# B&R Automation Studio project Soiled_PLC (part 5)

#### 12_sp2Cyclic.ab
```automation-basic
PROGRAM _CYCLIC
	(* cyclic program *)

;---------------------------------------
;Sequence 8 - SP8 Single point 2 D[912]
;---------------------------------------

;Inputs

O_SelectLine[11]          = FALSE
O_SelectLine[12]          = FALSE ;YB10
O_SelectLine[13]          = FALSE ;YB10
EnableRel.PC[2]           = FALSE
MySeq                     = 40
MyBag                     = 156
MyTransBag                = 158

I_BagatBuffer	          = RequestRel.PC[1]

O_Reset                   = FALSE

Alarm[MySeq].Name 			= 0
Alarm[MySeq].Bag			= MyTransBag
Alarm[MySeq].Beacon		    = TRUE
Alarm[MySeq].Extra			= 0
Alarm[MySeq].Time			= 5000

;Setup Sequence
STEP = D[900 + MySeq]
;Setup Pulse contact
PLS = (STEP <> LASTSTEP)
LASTSTEP = STEP

;Sequence
;Step 0 - Disabled
IF (STEP = 0) THEN
	;Disabled
ENDIF

;clear data
TON_10ms((STEP = 1),100,Reset,ResetET)
IF (STEP = 1) THEN
	O_Reset = TRUE
	IF (Reset = TRUE)AND (Bag[MyTransBag].Cat = 0) THEN
		D[900 + MySeq] = 2
	ENDIF
	IF Reset THEN
		Alarm[MySeq].Time			= 5
		Alarm[MySeq].Name 	= almBagDataError
	ENDIF
ENDIF

;Wait SLU1 request and destination clear
TON_10ms(I_BagatBuffer,300,BagAtBuffer,BagAtBufferET)
IF (STEP = 2) THEN
	IF (Bag[MyBag].Cat >0) AND (Bag[MyBag].Dst >0) AND RequestRel.PC[1] THEN
		IF (Line[Bag[MyBag].Dst].Space > 0) AND (Bag[MyBag].Dst > 10) AND (Bag[MyBag].Dst < 14) AND (Line[Bag[MyBag].Dst].Clear) AND (Bag[Line[Bag[MyBag].Dst].LastBag].Cat = 0) THEN
			Dest = Bag[MyBag].Dst
			C[Dest]        = 0
			D[900 + MySeq] = 3
		ENDIF

	ENDIF
ENDIF

		;Open buffer to release a bag to svc 1
IF (STEP = 3) THEN
	EnableRel.PC[2] = TRUE
	O_SelectLine[Dest] = TRUE
	IF PLS THEN
		IF (Bag[MyBag].Cat>0) AND (Bag[MyTransBag].Cat = 0)	THEN

			Bag[MyTransBag]     = Bag[MyBag]
			Bag[MyBag]          = Bag[0]
		ENDIF
	ENDIF
	IF (Dest = 13) THEN
		IF (Bag[MyTransBag].Cat>0) AND (Bag[159].Cat=0) AND X[4].X16 THEN
			Bag[159] = Bag[MyTransBag]
			Bag[MyTransBag] = Bag[0]
		ENDIF
		IF Line[Dest].Trip THEN
			IF ((Bag[73].Cat = 0) AND (Bag[159].Cat>0)) THEN
				Bag[159].Dst = 0
				Bag[73]      = Bag[159]
				Bag[159]     = Bag[0]
			ENDIF
			D[900 + MySeq] = 1
		ENDIF
    ELSE IF (Dest > 10) AND (Dest < 13) THEN
			IF Line[Dest].Trip THEN
				Bag[MyTransBag].Dst     = 0
				Bag[Line[Dest].LastBag] = Bag[MyTransBag]
				Bag[MyTransBag]         = Bag[0]
				D[900 + MySeq] = 1
		ENDIF

	ENDIF

	Alarm[MySeq].Name 	= almBagNotArrived
ENDIF

;select svc 2 point
IF (STEP = 4) THEN
O_SelectSVC2 = TRUE

	IF Line[18].Trip THEN
		IF (Bag[221].Cat > 0) AND (Bag[222].Cat= 0) THEN
			Bag[222] = Bag[221]
			Bag[221] = Bag[0]
		ENDIF
		D[900 + MySeq] = 1
	ENDIF
	Alarm[MySeq].Name 	= almBagNotArrived
ENDIF

;Outputs

Y[5].Y08 = O_SelectLine[11]
Y[5].Y09 = O_SelectLine[12]
Y[5].Y10 = O_Reset OR O_SelectLine[13]

;Alarms
TimerAlarm.IN 	= NOT PLS AND (Alarm[MySeq].Name > 0)
TimerAlarm.PT 	= Alarm[MySeq].Time
TimerAlarm FUB TON_10ms()
Alarm[MySeq].On 	= TimerAlarm.Q
Alarm[MySeq].ET 	= TimerAlarm.ET

;Outputs
;Y[6].Y07 = O_SelectPointSVC1
;Y[6].Y08 = O_SelectPointSVC2
END_PROGRAM
```

#### 12_sp2.var
```iecst
VAR RETAIN
	STEP : UINT;
	PLS : BOOL;
	LASTSTEP : UINT;
END_VAR
VAR
	TimerAlarm : TON_10ms;
	I_BagAtBuffer : BOOL;
	O_OpenBuffer : BOOL;
	SDC2BufferFullET : TIME;
	SDC2BufferFull : BOOL;
	SettledBufferET : TIME;
	SettledBuffer : BOOL;
	O_OpenSP2BufferStop : BOOL;
	O_SelectPoint : BOOL;
	SP2BufferFull : BOOL;
	SP2BufferFullET : UDINT;
	ParingLoopEnabled : BOOL;
	BagInLoopHasDest : BOOL;
	BagAtBuffer : BOOL;
	SettledBufferSVC1 : BOOL;
	SettledBufferSVC1ET : UDINT;
	SettledBufferSVC2 : BOOL;
	SettledBufferSVC2ET : UDINT;
	O_SelectPointSVC1 : BOOL;
	O_SelectPointSVC2 : BOOL;
	Reset : BOOL;
	ResetET : UDINT;
	I_BagatBuffer : BOOL;
	BagAtBufferET : UDINT;
	Alernate : USINT;
	I_BagAtSVC1BufferStop : BOOL;
	O_SVC1BufferStop : BOOL;
	I_BagAtSVC2BufferStop : BOOL;
	O_SVC2BufferStop : BOOL;
	O_SelectSVC1 : BOOL;
	O_SelectSVC2 : BOOL;
	MySeq : USINT;
	MyBag : USINT;
	MyTransBag : INT;
	Dest : INT;
	O_SelectLine : ARRAY[0..13] OF BOOL;
	O_Reset : BOOL;
END_VAR
```

### Program Logical/Sequences/10ms/41_cp8 (IEC) - * SP2 Empty bags from SDC1/2

#### 12_sp2.var
```iecst
VAR RETAIN
	STEP : UINT;
	PLS : BOOL;
	LASTSTEP : UINT;
END_VAR
VAR
	TimerAlarm : TON_10ms;
	I_BagAtBuffer : ARRAY[0..3] OF BOOL;
	O_OpenBuffer : BOOL;
	SDC2BufferFullET : TIME;
	SDC2BufferFull : BOOL;
	SettledBufferET : TIME;
	SettledBuffer : ARRAY[0..3] OF BOOL;
	O_OpenSP2BufferStop : BOOL;
	O_SelectPoint : BOOL;
	SP2BufferFull : BOOL;
	SP2BufferFullET : UDINT;
	ParingLoopEnabled : BOOL;
	BagInLoopHasDest : BOOL;
	O_OpenSDC1BufferStop : BOOL;
	BagSettledAtBuffer : BOOL;
	BagSettledAtBufferET : UDINT;
	Alternator : USINT;
	I_OnLineA : BOOL;
	I_TiltA : BOOL;
	I_TiltB : BOOL;
	I_Bagout : BOOL;
	O_OpenBufferStop : BOOL;
	O_SelectLineA : BOOL;
	O_SelectLineB : BOOL;
	O_OpenStops : BOOL;
	O_TiltCylinder : BOOL;
	O_OperatePusher : BOOL;
	PointReset : BOOL;
	PointResetET : UDINT;
	BagAtTilt : BOOL;
	BagAtTiltET : UDINT;
	TiltDown : BOOL;
	TiltDownET : UDINT;
	TiltUp : BOOL;
	TiltUpET : UDINT;
	NotFull : BOOL;
	NotFullET : UDINT;
	Pushed : BOOL;
	SBSN1 : BOOL;
	SBSN1ET : UDINT;
	RequirePusherET : UDINT;
	PushedET : UDINT;
	I_BagAtBufferStop : BOOL;
	O_SP7ToSVC1 : BOOL;
	O_SP7ToSIC3 : BOOL;
	SDC1EmptyBufferFull : BOOL;
	SDC1EmptyBufferFullET : UDINT;
	Reset : BOOL;
	ResetET : UDINT;
	ResetPoint : BOOL;
	I_SDC1EmptyBagAtBuffer : BOOL;
	O_ResetPoints : BOOL;
	BagSettledSDC1Buffer : BOOL;
	BagSettledSDC1BufferET : UDINT;
	BagSettledSDC2Buffer : BOOL;
	BagSettledSDC2BufferET : UDINT;
	MySeq : USINT;
	BagSettledBufferET : ARRAY[0..3] OF UDINT;
	Alt : USINT;
	O_SelectCDC4 : BOOL;
	O_SelectStraight : BOOL;
	O_SelectCDC3 : BOOL;
	O_SelectCPI4 : BOOL;
	O_SelectCP6 : BOOL;
	O_Reset : BOOL;
END_VAR
```

#### 12_sp2Cyclic.ab
```automation-basic
PROGRAM _CYCLIC
	(* cyclic program *)

;---------------------------------------
;Sequence 12 - SP2 Single point 2 D[912]
;---------------------------------------

;Inputs

I_BagAtBuffer[1]		= Request.DCEmptyRelease[3]
I_BagAtBuffer[2]		= X[10].X04
I_BagAtBuffer[3]		= X[10].X05

MySeq                   = 41

Alarm[MySeq].Name 			= 0
Alarm[MySeq].Bag			= 10013
Alarm[MySeq].Beacon		= TRUE
Alarm[MySeq].Extra			= 0
Alarm[MySeq].Time			= 3000

Enable.DCEmptyRelease[3]    = FALSE

O_SelectCDC3                = FALSE
O_SelectCPI4                = FALSE
O_SelectCP6                 = FALSE
O_Reset                     = FALSE

;Setup Sequence
STEP = D[900 + MySeq]
;Setup Pulse contact
PLS = (STEP <> LASTSTEP)
LASTSTEP = STEP

;Sequence
;Step 0 - Disabled
IF (STEP = 0) THEN
	;Disabled
ENDIF

;reset points
TON_10ms((STEP = 1),200,Reset,ResetET)
IF (STEP = 1) THEN
	O_Reset = NOT Reset
	IF (Line[42].Clear) AND Reset  THEN
		D[900 + MySeq] = 2
	ENDIF
	ELSE

ENDIF

;check which bag is ready
TON_10ms(I_BagAtBuffer[1],200,SettledBuffer[1],BagSettledBufferET[1])
TON_10ms(I_BagAtBuffer[2],200,SettledBuffer[2],BagSettledBufferET[2])
TON_10ms(I_BagAtBuffer[3],200,SettledBuffer[3],BagSettledBufferET[3])
IF (STEP = 2) THEN
	IF (Line[42].Clear) AND NOT Y[4].Y15 AND NOT X[8].X08 THEN
		;Alt = Alt + 1
		;IF (Alt > 2) THEN
		;	Alt = 0
		;ENDIF
		IF SettledBuffer[1]  THEN
			C[42]          = 0
		    D[900 + MySeq] = 3
		ELSE IF SettledBuffer[2]  THEN
			C[42]          = 0
			D[900 + MySeq] = 4
		ELSE IF SettledBuffer[3] AND (D[8]>0)  THEN
			C[42]          = 0
			D[900 + MySeq] = 5
		ENDIF
	ENDIF
ENDIF

;Bag at line
IF (STEP = 3) THEN
	O_SelectCDC3 = TRUE
	Enable.DCEmptyRelease[3] = TRUE
	IF (Line[42].Trip = TRUE) THEN
		D[900 + MySeq] = 1
	ENDIF
	Alarm[MySeq].Name 	  = almBagNotArrived
ENDIF

;Bag at line
IF (STEP = 4) THEN
	O_SelectCP6 = TRUE
	IF (Line[42].Trip = TRUE) THEN
		D[900 + MySeq] = 1
	ENDIF
	Alarm[MySeq].Name 	  = almBagNotArrived
ENDIF

;Bag at line
IF (STEP = 5) THEN
	O_SelectCPI4 = TRUE
	IF (Line[42].Trip = TRUE) THEN
		D[900 + MySeq] = 1
	ENDIF
	Alarm[MySeq].Name 	  = almBagNotArrived
ENDIF
;Alarms
TimerAlarm.IN 	= NOT PLS AND (Alarm[MySeq].Name > 0)
TimerAlarm.PT 	= Alarm[MySeq].Time
TimerAlarm FUB TON_10ms()
Alarm[MySeq].On 	= TimerAlarm.Q
Alarm[MySeq].ET 	= TimerAlarm.ET

;Outputs
Y[9].Y09 = O_SelectCDC3
Y[8].Y03 = O_SelectCP6
Y[8].Y04 = O_SelectCPI4
Y[8].Y08 = O_Reset

END_PROGRAM
```

### Program Logical/Sequences/10ms/42_cp9 (IEC) - * SP2 Empty bags from SDC1/2

#### 12_sp2.var
```iecst
VAR RETAIN
	STEP : UINT;
	PLS : BOOL;
	LASTSTEP : UINT;
END_VAR
VAR
	TimerAlarm : TON_10ms;
	I_BagAtBuffer : ARRAY[0..3] OF BOOL;
	O_OpenBuffer : BOOL;
	SDC2BufferFullET : TIME;
	SDC2BufferFull : BOOL;
	SettledBufferET : TIME;
	SettledBuffer : ARRAY[0..3] OF BOOL;
	O_OpenSP2BufferStop : BOOL;
	O_SelectPoint : BOOL;
	SP2BufferFull : BOOL;
	SP2BufferFullET : UDINT;
	ParingLoopEnabled : BOOL;
	BagInLoopHasDest : BOOL;
	O_OpenSDC1BufferStop : BOOL;
	BagSettledAtBuffer : BOOL;
	BagSettledAtBufferET : UDINT;
	Alternator : USINT;
	I_OnLineA : BOOL;
	I_TiltA : BOOL;
	I_TiltB : BOOL;
	I_Bagout : BOOL;
	O_OpenBufferStop : BOOL;
	O_SelectLineA : BOOL;
	O_SelectLineB : BOOL;
	O_OpenStops : BOOL;
	O_TiltCylinder : BOOL;
	O_OperatePusher : BOOL;
	PointReset : BOOL;
	PointResetET : UDINT;
	BagAtTilt : BOOL;
	BagAtTiltET : UDINT;
	TiltDown : BOOL;
	TiltDownET : UDINT;
	TiltUp : BOOL;
	TiltUpET : UDINT;
	NotFull : BOOL;
	NotFullET : UDINT;
	Pushed : BOOL;
	SBSN1 : BOOL;
	SBSN1ET : UDINT;
	RequirePusherET : UDINT;
	PushedET : UDINT;
	I_BagAtBufferStop : BOOL;
	O_SP7ToSVC1 : BOOL;
	O_SP7ToSIC3 : BOOL;
	SDC1EmptyBufferFull : BOOL;
	SDC1EmptyBufferFullET : UDINT;
	Reset : BOOL;
	ResetET : UDINT;
	ResetPoint : BOOL;
	I_SDC1EmptyBagAtBuffer : BOOL;
	O_ResetPoints : BOOL;
	BagSettledSDC1Buffer : BOOL;
	BagSettledSDC1BufferET : UDINT;
	BagSettledSDC2Buffer : BOOL;
	BagSettledSDC2BufferET : UDINT;
	MySeq : USINT;
	BagSettledBufferET : ARRAY[0..3] OF UDINT;
	Alt : USINT;
	O_SelectCDC4 : BOOL;
	O_SelectStraight : BOOL;
	O_Reset : BOOL;
	O_SelectCLU1 : BOOL;
	O_SelectCLU2 : BOOL;
END_VAR
```

#### 12_sp2Cyclic.ab
```automation-basic
PROGRAM _CYCLIC
	(* cyclic program *)

;---------------------------------------
;Sequence 12 - SP2 Single point 2 D[912]
;---------------------------------------

;Inputs

I_BagAtBuffer[1]		= X[8].X16
;I_BagAtBuffer[2]		= X[9].X14

MySeq                   = 42

Alarm[MySeq].Name 			= 0
Alarm[MySeq].Bag			= 10005
Alarm[MySeq].Beacon		= TRUE
Alarm[MySeq].Extra			= 0
Alarm[MySeq].Time			= 3000

O_SelectCLU1                = FALSE
O_SelectCLU2                = FALSE

;Setup Sequence
STEP = D[900 + MySeq]
;Setup Pulse contact
PLS = (STEP <> LASTSTEP)
LASTSTEP = STEP

;Sequence
;Step 0 - Disabled
IF (STEP = 0) THEN
	;Disabled
ENDIF

;reset points
TON_10ms((STEP = 1),200,Reset,ResetET)
IF (STEP = 1) THEN
	O_Reset = NOT Reset
	IF (Reset)  THEN
		D[900 + MySeq] = 2
	ENDIF
	ELSE

ENDIF

;check which bag is ready
TON_10ms(I_BagAtBuffer[1],200,SettledBuffer[1],BagSettledBufferET[1])

IF (STEP = 2) THEN
	IF SettledBuffer[1] THEN
		Alt = Alt + 1
		IF (Alt > 2) THEN
			Alt = 0
		ENDIF
		IF SettledBuffer[1] AND (Alt = 1) AND Line[35].Clear THEN
			C[35]          = 0
		    D[900 + MySeq] = 3
		ELSE IF SettledBuffer[1] AND (Alt = 2) AND Line[36].Clear THEN
			C[36]          = 0
			D[900 + MySeq] = 4
		ENDIF
	ENDIF
ENDIF

;Bag at line
IF (STEP = 3) THEN
	O_SelectCLU1 = TRUE
	IF (Line[35].Trip = TRUE) THEN
		D[900 + MySeq] = 1
	ENDIF
	Alarm[MySeq].Name 	  = almBagNotArrived
ENDIF

;Bag at line
IF (STEP = 4) THEN
	O_SelectCLU2 = TRUE
	IF (Line[36].Trip = TRUE) THEN
		D[900 + MySeq] = 1
	ENDIF
	Alarm[MySeq].Name 	  = almBagNotArrived
ENDIF

;Alarms
TimerAlarm.IN 	= NOT PLS AND (Alarm[MySeq].Name > 0)
TimerAlarm.PT 	= Alarm[MySeq].Time
TimerAlarm FUB TON_10ms()
Alarm[MySeq].On 	= TimerAlarm.Q
Alarm[MySeq].ET 	= TimerAlarm.ET

;Outputs
Y[8].Y05 = O_SelectCLU1
Y[8].Y06 = O_SelectCLU2
Y[8].Y07 = O_SelectCLU1 OR O_SelectCLU2
END_PROGRAM
```

### Program Logical/Sequences/10ms/43_cp12 (IEC) - * SP2 Empty bags from SDC1/2

#### 12_sp2.var
```iecst
VAR RETAIN
	STEP : UINT;
	PLS : BOOL;
	LASTSTEP : UINT;
END_VAR
VAR
	TimerAlarm : TON_10ms;
	I_BagAtBuffer : ARRAY[0..3] OF BOOL;
	O_OpenBuffer : BOOL;
	SDC2BufferFullET : TIME;
	SDC2BufferFull : BOOL;
	SettledBufferET : TIME;
	SettledBuffer : ARRAY[0..3] OF BOOL;
	O_OpenSP2BufferStop : BOOL;
	O_SelectPoint : BOOL;
	SP2BufferFull : BOOL;
	SP2BufferFullET : UDINT;
	ParingLoopEnabled : BOOL;
	BagInLoopHasDest : BOOL;
	O_OpenSDC1BufferStop : BOOL;
	BagSettledAtBuffer : BOOL;
	BagSettledAtBufferET : UDINT;
	Alternator : USINT;
	I_OnLineA : BOOL;
	I_TiltA : BOOL;
	I_TiltB : BOOL;
	I_Bagout : BOOL;
	O_OpenBufferStop : BOOL;
	O_SelectLineA : BOOL;
	O_SelectLineB : BOOL;
	O_OpenStops : BOOL;
	O_TiltCylinder : BOOL;
	O_OperatePusher : BOOL;
	PointReset : BOOL;
	PointResetET : UDINT;
	BagAtTilt : BOOL;
	BagAtTiltET : UDINT;
	TiltDown : BOOL;
	TiltDownET : UDINT;
	TiltUp : BOOL;
	TiltUpET : UDINT;
	NotFull : BOOL;
	NotFullET : UDINT;
	Pushed : BOOL;
	SBSN1 : BOOL;
	SBSN1ET : UDINT;
	RequirePusherET : UDINT;
	PushedET : UDINT;
	I_BagAtBufferStop : BOOL;
	O_SP7ToSVC1 : BOOL;
	O_SP7ToSIC3 : BOOL;
	SDC1EmptyBufferFull : BOOL;
	SDC1EmptyBufferFullET : UDINT;
	Reset : BOOL;
	ResetET : UDINT;
	ResetPoint : BOOL;
	I_SDC1EmptyBagAtBuffer : BOOL;
	O_ResetPoints : BOOL;
	BagSettledSDC1Buffer : BOOL;
	BagSettledSDC1BufferET : UDINT;
	BagSettledSDC2Buffer : BOOL;
	BagSettledSDC2BufferET : UDINT;
	MySeq : USINT;
	BagSettledBufferET : ARRAY[0..3] OF UDINT;
	Alt : USINT;
	O_SelectCDC4 : BOOL;
	O_SelectStraight : BOOL;
	O_SelectCIC5 : BOOL;
	O_SelectCDC6 : BOOL;
	O_Reset : BOOL;
	O_SelectCDC5 : BOOL;
	O_SelectCDC7 : BOOL;
	O_SelectCDC8 : BOOL;
	O_SelectCDC9 : BOOL;
	Dest : USINT;
END_VAR
```

#### 12_sp2Cyclic.ab
```automation-basic
PROGRAM _CYCLIC
	(* cyclic program *)

;---------------------------------------
;Sequence 12 - SP2 Single point 2 D[912]
;---------------------------------------

;Inputs

I_BagAtBuffer[1]		= RequestRel.IC[5]
;I_BagAtBuffer[2]		= X[9].X14

MySeq                   = 43

Alarm[MySeq].Name 			= 0
Alarm[MySeq].Bag			= 166
Alarm[MySeq].Beacon		= TRUE
Alarm[MySeq].Extra			= 0
Alarm[MySeq].Time			= 3000

O_SelectCDC7                = FALSE
O_SelectCDC8               = FALSE
O_SelectCDC9                = FALSE
EnableRel.IC[5]             = FALSE
O_Reset                     = FALSE

;Setup Sequence
STEP = D[900 + MySeq]
;Setup Pulse contact
PLS = (STEP <> LASTSTEP)
LASTSTEP = STEP

;Sequence
;Step 0 - Disabled
IF (STEP = 0) THEN
	;Disabled
ENDIF

;reset points
TON_10ms((STEP = 1),200,Reset,ResetET)
IF (STEP = 1) THEN
	O_Reset = TRUE
	IF Reset  THEN
		D[900 + MySeq] = 2
	ENDIF
	ELSE

ENDIF

;check which bag is ready
TON_10ms(I_BagAtBuffer[1],200,SettledBuffer[1],BagSettledBufferET[1])

IF (STEP = 2) THEN
	IF SettledBuffer[1] AND (D[43] >0)  THEN
		Dest = Bag[152].Dst
		IF (Dest = 17) AND Line[17].Clear AND (Bag[92].Cat = 0) THEN
			C[17]                  = 0
			D[900 + MySeq] = 3
        ELSE IF (Dest = 18) AND Line[18].Clear AND (Bag[97].Cat = 0) THEN
			C[18]                  = 0
			D[900 + MySeq] = 4
		 ELSE IF (Dest = 19) AND Line[26].Clear AND (Bag[151].Cat = 0) THEN
			C[26]                  = 0
			D[900 + MySeq] = 5
		ENDIF
	ENDIF
ENDIF

;Bag at line
IF (STEP = 3) THEN
	O_SelectCDC7 = TRUE
	EnableRel.IC[5] = TRUE
;	IF (Bag[152].Cat>0) AND (Bag[166].Cat = 0) THEN
;		Bag[166] = Bag[152]
;		Bag[152] = Bag[0]
;	ENDIF
	IF Line[17].Trip THEN
		IF (Bag[166].Cat > 0) AND (Bag[92].Cat = 0) THEN
			Bag[92] = Bag[166]
			Bag[166]= Bag[0]

		ENDIF
			D[900 + MySeq] = 1
	ENDIF
	Alarm[MySeq].Name 	  = almBagNotArrived
ENDIF

;Bag at line
IF (STEP = 4) THEN
	O_SelectCDC8 = TRUE
	EnableRel.IC[5] = TRUE
;	IF (Bag[152].Cat>0) AND (Bag[166].Cat = 0) THEN
;		Bag[166] = Bag[152]
;		Bag[152] = Bag[0]
;	ENDIF
	IF (Line[18].Trip = TRUE) THEN
		IF (Bag[166].Cat > 0) AND (Bag[97].Cat = 0) THEN
			Bag[97] = Bag[166]
			Bag[166]= Bag[0]

		ENDIF
		D[900 + MySeq] = 1
	ENDIF
	Alarm[MySeq].Name 	  = almBagNotArrived
ENDIF

IF (STEP = 5) THEN
	O_SelectCDC9 = TRUE
	EnableRel.IC[5] = TRUE
;	IF (Bag[152].Cat>0) AND (Bag[166].Cat = 0) THEN
;		Bag[166] = Bag[152]
;		Bag[152] = Bag[0]
;	ENDIF
	IF (Line[26].Trip = TRUE) THEN
		IF (Bag[166].Cat > 0) AND (Bag[151].Cat = 0) THEN
			Bag[166].Dst = 0
			Bag[151]       = Bag[166]
			Bag[166]       = Bag[0]

		ENDIF
		D[900 + MySeq] = 1
	ENDIF
	Alarm[MySeq].Name 	  = almBagNotArrived
ENDIF

;Alarms
TimerAlarm.IN 	= NOT PLS AND (Alarm[MySeq].Name > 0)
TimerAlarm.PT 	= Alarm[MySeq].Time
TimerAlarm FUB TON_10ms()
Alarm[MySeq].On 	= TimerAlarm.Q
Alarm[MySeq].ET 	= TimerAlarm.ET

;Outputs
Y[1].Y13 = O_SelectCDC7
Y[2].Y03 = O_SelectCDC8
Y[10].Y03 = O_Reset OR O_SelectCDC9
Y[10].Y04 = O_Reset OR O_SelectCDC9
END_PROGRAM
```

### Program Logical/Sequences/10ms/44_cpr2 (IEC, version 1.00.2) - *Pressure Relief

#### pr.st - Implementation code
```iecst
(********************************************************************
 * COPYRIGHT --
 ********************************************************************
 * Program: pr
 * File: pr.st
 * Author: treamsbottom
 * Created: July 16, 2015
 ********************************************************************
 * Implementation of program pr
 ********************************************************************)

PROGRAM _INIT
//Configuration
mySeq						:= 44;	//Sequence number
myIO						:= 9;
myZone						:= 0;
myRelLine					:= 28;
myBag						:= 0; //Buffer Bag
bufferSettleTime			:= 300;

myOutBag 					:= Line[myRelLine].LastBag;
END_PROGRAM

PROGRAM _CYCLIC
//Inputs
i_bagAtBuffer				:= X[myIO].X08;

i_bagAtBufferOut 		:= FALSE; // Any Single bag buffer out IO.
i_bufferOutOpen			:= FALSE;

o_openBuffer	:= FALSE;

IF (myBag = 0) THEN
	Alarm[mySeq].Bag	:= mySeq + 10000;
ELSE
	Alarm[mySeq].Bag	:= myBag;
END_IF;

Alarm[mySeq].Name 		:= 0;
Alarm[mySeq].Beacon		:= TRUE;
Alarm[mySeq].Extra		:= 0;
Alarm[mySeq].Time		:= 3000;

//Setup Sequence
step := D[900 + mySeq];
//Setup Pulse contact
pls := (step <> lastStep);
lastStep := step;

//Sequence
IF (step = 0) THEN
	//Disabled
END_IF;

//Bag Settled at buffer
ton_10ms_SettledBuffer(IN:= i_bagAtBuffer, PT:= bufferSettleTime);
IF (step = 1) THEN
	IF ton_10ms_SettledBuffer.Q AND NOT Std.HaltSysZone[myZone]THEN
		IF Line[myRelLine].Clear AND NOT i_bagAtBufferOut AND NOT i_bufferOutOpen AND NOT Line[myRelLine].Trip THEN
			IF (myBag = 0) THEN
				C[myRelLine] := 0;
				D[900 + mySeq] := 2;
			ELSIF (Bag[myBag].Cat > 0) AND (Bag[myOutBag].Cat = 0) THEN
				C[myRelLine] := 0;
				D[900 + mySeq] := 2;
			ELSIF (Bag[myBag].Cat = 0) THEN
				Alarm[mySeq].Name := ALM_BAG_DATA_ERROR;
				Alarm[mySeq].Time := 0;
			ELSIF (Bag[myOutBag].Cat > 0) THEN
				Alarm[mySeq].Name := ALM_BAG_DATA_ERROR;
				Alarm[mySeq].Bag := myOutBag;
				Alarm[mySeq].Time := 0;
			END_IF;
		ELSIF Line[myRelLine].Trip THEN
			Alarm[mySeq].Name := ALM_SWITCH_FAULT; //Trip is stuck on
			Alarm[mySeq].Time := 500;
		END_IF;
	ELSIF (myBag > 0) AND (Bag[myBag].Cat > 0) THEN
		Alarm[mySeq].Name := ALM_BAG_NOT_SETTLED;
	END_IF;
END_IF;

IF (step = 2) THEN
	dataValid := ((myBag = 0) OR ((Bag[myBag].Cat > 0) AND (Bag[myOutBag].Cat = 0)));
	o_openBuffer :=  dataValid;
	IF dataValid THEN
		IF Line[myRelLine].Trip THEN
			IF (myBag > 0) THEN
				Bag[myOutBag] := Bag[myBag];
				Bag[myBag]  := Bag[0];
			END_IF;
			D[900 + mySeq] := 1;
		END_IF;
		Alarm[mySeq].Name := ALM_BAG_NOT_RELEASED;
	ELSIF (myBag > 0) THEN
		IF (Bag[myBag].Cat = 0) THEN
			Alarm[mySeq].Name := ALM_BAG_DATA_ERROR;
			Alarm[mySeq].Time := 0;
		ELSIF (Bag[myOutBag].Cat > 0) THEN
			Alarm[mySeq].Name := ALM_BAG_DATA_ERROR;
			Alarm[mySeq].Bag := myOutBag;
			Alarm[mySeq].Time := 0;
		END_IF;
	END_IF;
END_IF;

//-----------------------------------
//PLC Outputs - adjust TO suit system
//-----------------------------------

Y[myIO].Y08 := o_openBuffer;

//Alarms
timerAlarm(IN := NOT pls AND (Alarm[mySeq].Name > 0),PT:= Alarm[mySeq].Time);

Alarm[mySeq].On 	:= timerAlarm.Q;
Alarm[mySeq].ET 	:= timerAlarm.ET;

END_PROGRAM
```

### Program Logical/Sequences/10ms/45_cpr3 (IEC) - *Pressure Relief

#### pr.st
```iecst
(********************************************************************
 * COPYRIGHT --
 ********************************************************************
 * Program: pr
 * File: pr.st
 * Author: treamsbottom
 * Created: July 16, 2015
 ********************************************************************
 * Implementation of program pr
 ********************************************************************)

PROGRAM _INIT
//Configuration
mySeq						:= 45;	//Sequence number
myIO						:= 9;
myZone						:= 0;
myRelLine					:= 39;
myBag						:= 0; //Buffer Bag
bufferSettleTime			:= 300;

myOutBag 					:= Line[myRelLine].LastBag;
END_PROGRAM

PROGRAM _CYCLIC
//Inputs
i_bagAtBuffer				:= X[myIO].X12;

i_bagAtBufferOut 		:= FALSE; // Any Single bag buffer out IO.
i_bufferOutOpen			:= FALSE;

o_openBuffer	:= FALSE;

IF (myBag = 0) THEN
	Alarm[mySeq].Bag	:= mySeq + 10000;
ELSE
	Alarm[mySeq].Bag	:= myBag;
END_IF;

Alarm[mySeq].Name 		:= 0;
Alarm[mySeq].Beacon		:= TRUE;
Alarm[mySeq].Extra		:= 0;
Alarm[mySeq].Time		:= 3000;

//Setup Sequence
step := D[900 + mySeq];
//Setup Pulse contact
pls := (step <> lastStep);
lastStep := step;

//Sequence
IF (step = 0) THEN
	//Disabled
END_IF;

//Bag Settled at buffer
ton_10ms_SettledBuffer(IN:= i_bagAtBuffer, PT:= bufferSettleTime);
IF (step = 1) THEN
	IF ton_10ms_SettledBuffer.Q AND NOT Std.HaltSysZone[myZone]THEN
		IF Line[myRelLine].Clear AND NOT i_bagAtBufferOut AND NOT i_bufferOutOpen AND NOT Line[myRelLine].Trip THEN
			IF (myBag = 0) THEN
				C[myRelLine] := 0;
				D[900 + mySeq] := 2;
			ELSIF (Bag[myBag].Cat > 0) AND (Bag[myOutBag].Cat = 0) THEN
				C[myRelLine] := 0;
				D[900 + mySeq] := 2;
			ELSIF (Bag[myBag].Cat = 0) THEN
				Alarm[mySeq].Name := ALM_BAG_DATA_ERROR;
				Alarm[mySeq].Time := 0;
			ELSIF (Bag[myOutBag].Cat > 0) THEN
				Alarm[mySeq].Name := ALM_BAG_DATA_ERROR;
				Alarm[mySeq].Bag := myOutBag;
				Alarm[mySeq].Time := 0;
			END_IF;
		ELSIF Line[myRelLine].Trip THEN
			Alarm[mySeq].Name := ALM_SWITCH_FAULT; //Trip is stuck on
			Alarm[mySeq].Time := 500;
		END_IF;
	ELSIF (myBag > 0) AND (Bag[myBag].Cat > 0) THEN
		Alarm[mySeq].Name := ALM_BAG_NOT_SETTLED;
	END_IF;
END_IF;

IF (step = 2) THEN
	dataValid := ((myBag = 0) OR ((Bag[myBag].Cat > 0) AND (Bag[myOutBag].Cat = 0)));
	o_openBuffer :=  dataValid;
	IF dataValid THEN
		IF Line[myRelLine].Trip THEN
			IF (myBag > 0) THEN
				Bag[myOutBag] := Bag[myBag];
				Bag[myBag]  := Bag[0];
			END_IF;
			D[900 + mySeq] := 1;
		END_IF;
		Alarm[mySeq].Name := ALM_BAG_NOT_RELEASED;
	ELSIF (myBag > 0) THEN
		IF (Bag[myBag].Cat = 0) THEN
			Alarm[mySeq].Name := ALM_BAG_DATA_ERROR;
			Alarm[mySeq].Time := 0;
		ELSIF (Bag[myOutBag].Cat > 0) THEN
			Alarm[mySeq].Name := ALM_BAG_DATA_ERROR;
			Alarm[mySeq].Bag := myOutBag;
			Alarm[mySeq].Time := 0;
		END_IF;
	END_IF;
END_IF;

//-----------------------------------
//PLC Outputs - adjust TO suit system
//-----------------------------------

Y[9].Y12 := o_openBuffer;

//Alarms
timerAlarm(IN := NOT pls AND (Alarm[mySeq].Name > 0),PT:= Alarm[mySeq].Time);

Alarm[mySeq].On 	:= timerAlarm.Q;
Alarm[mySeq].ET 	:= timerAlarm.ET;

END_PROGRAM
```

### Program Logical/Sequences/10ms/46_cpr4 (IEC) - *Pressure Relief

#### pr.st
```iecst
(********************************************************************
 * COPYRIGHT --
 ********************************************************************
 * Program: pr
 * File: pr.st
 * Author: treamsbottom
 * Created: July 16, 2015
 ********************************************************************
 * Implementation of program pr
 ********************************************************************)

PROGRAM _INIT
//Configuration
mySeq						:= 46;	//Sequence number
myIO						:= 220;
myZone						:= 0;
myRelLine					:= 40;
myBag						:= 0; //Buffer Bag
bufferSettleTime			:= 300;

myOutBag 					:= Line[myRelLine].LastBag;
END_PROGRAM

PROGRAM _CYCLIC
//Inputs
i_bagAtBuffer				:= X[11].X10;

i_bagAtBufferOut 		:= FALSE; // Any Single bag buffer out IO.
i_bufferOutOpen			:= FALSE;

o_openBuffer	:= FALSE;

IF (myBag = 0) THEN
	Alarm[mySeq].Bag	:= mySeq + 10000;
ELSE
	Alarm[mySeq].Bag	:= myBag;
END_IF;

Alarm[mySeq].Name 		:= 0;
Alarm[mySeq].Beacon		:= TRUE;
Alarm[mySeq].Extra		:= 0;
Alarm[mySeq].Time		:= 3000;

//Setup Sequence
step := D[900 + mySeq];
//Setup Pulse contact
pls := (step <> lastStep);
lastStep := step;

//Sequence
IF (step = 0) THEN
	//Disabled
END_IF;

//Bag Settled at buffer
ton_10ms_SettledBuffer(IN:= i_bagAtBuffer, PT:= bufferSettleTime);
IF (step = 1) THEN
	IF ton_10ms_SettledBuffer.Q AND NOT Std.HaltSysZone[myZone]THEN
		IF Line[myRelLine].Clear AND NOT i_bagAtBufferOut AND NOT i_bufferOutOpen AND NOT Line[myRelLine].Trip THEN
			IF (myBag = 0) THEN
				C[myRelLine] := 0;
				D[900 + mySeq] := 2;
			ELSIF (Bag[myBag].Cat > 0) AND (Bag[myOutBag].Cat = 0) THEN
				C[myRelLine] := 0;
				D[900 + mySeq] := 2;
			ELSIF (Bag[myBag].Cat = 0) THEN
				Alarm[mySeq].Name := ALM_BAG_DATA_ERROR;
				Alarm[mySeq].Time := 0;
			ELSIF (Bag[myOutBag].Cat > 0) THEN
				Alarm[mySeq].Name := ALM_BAG_DATA_ERROR;
				Alarm[mySeq].Bag := myOutBag;
				Alarm[mySeq].Time := 0;
			END_IF;
		ELSIF Line[myRelLine].Trip THEN
			Alarm[mySeq].Name := ALM_SWITCH_FAULT; //Trip is stuck on
			Alarm[mySeq].Time := 500;
		END_IF;
	ELSIF (myBag > 0) AND (Bag[myBag].Cat > 0) THEN
		Alarm[mySeq].Name := ALM_BAG_NOT_SETTLED;
	END_IF;
END_IF;

IF (step = 2) THEN
	dataValid := ((myBag = 0) OR ((Bag[myBag].Cat > 0) AND (Bag[myOutBag].Cat = 0)));
	o_openBuffer :=  dataValid;
	IF dataValid THEN
		IF Line[myRelLine].Trip THEN
			IF (myBag > 0) THEN
				Bag[myOutBag] := Bag[myBag];
				Bag[myBag]  := Bag[0];
			END_IF;
			D[900 + mySeq] := 1;
		END_IF;
		Alarm[mySeq].Name := ALM_BAG_NOT_RELEASED;
	ELSIF (myBag > 0) THEN
		IF (Bag[myBag].Cat = 0) THEN
			Alarm[mySeq].Name := ALM_BAG_DATA_ERROR;
			Alarm[mySeq].Time := 0;
		ELSIF (Bag[myOutBag].Cat > 0) THEN
			Alarm[mySeq].Name := ALM_BAG_DATA_ERROR;
			Alarm[mySeq].Bag := myOutBag;
			Alarm[mySeq].Time := 0;
		END_IF;
	END_IF;
END_IF;

//-----------------------------------
//PLC Outputs - adjust TO suit system
//-----------------------------------

Y[10].Y10 := o_openBuffer;

//Alarms
timerAlarm(IN := NOT pls AND (Alarm[mySeq].Name > 0),PT:= Alarm[mySeq].Time);

Alarm[mySeq].On 	:= timerAlarm.Q;
Alarm[mySeq].ET 	:= timerAlarm.ET;

END_PROGRAM
```

- Standard_Sequence_Pressure_Relief_ENG.docx (binary file, 203948 bytes)
### Program Logical/Sequences/10ms/47_cpr1 (IEC) - *Pressure Relief

#### pr.var
```iecst
(********************************************************************
 * COPYRIGHT --
 ********************************************************************
 * Program: pr
 * File: pr.var
 * Author: treamsbottom
 * Created: July 16, 2015
 ********************************************************************
 * Local variables of program pr
 ********************************************************************)
VAR
	mySeq : UINT;
	myIO : UINT;
	myZone : UINT;
	myRelLine : UINT;
	myBag : UINT;
	i_bagAtBuffer : BOOL;
	i_bagAtBufferOut : BOOL;
	i_bufferOutOpen : BOOL;
	o_openBuffer : BOOL;
	step : UINT;
	pls : BOOL;
	timerAlarm : TON_10ms;
END_VAR
VAR RETAIN
	lastStep : UINT;
END_VAR
VAR
	bufferSettleTime : UDINT;
	ton_10ms_SettledBuffer : TON_10ms;
	myOutBag : UINT;
	dataValid : BOOL;
END_VAR
```

#### pr.st
```iecst
(********************************************************************
 * COPYRIGHT --
 ********************************************************************
 * Program: pr
 * File: pr.st
 * Author: treamsbottom
 * Created: July 16, 2015
 ********************************************************************
 * Implementation of program pr
 ********************************************************************)

PROGRAM _INIT
//Configuration
mySeq						:= 47;	//Sequence number
myIO						:= 9;
myZone						:= 0;
myRelLine					:= 43;
myBag						:= 0; //Buffer Bag
bufferSettleTime			:= 300;

myOutBag 					:= Line[myRelLine].LastBag;
END_PROGRAM

PROGRAM _CYCLIC
//Inputs
i_bagAtBuffer				:= X[myIO].X03;

i_bagAtBufferOut 		:= FALSE; // Any Single bag buffer out IO.
i_bufferOutOpen			:= FALSE;

o_openBuffer	:= FALSE;

IF (myBag = 0) THEN
	Alarm[mySeq].Bag	:= mySeq + 10000;
ELSE
	Alarm[mySeq].Bag	:= myBag;
END_IF;

Alarm[mySeq].Name 		:= 0;
Alarm[mySeq].Beacon		:= TRUE;
Alarm[mySeq].Extra		:= 0;
Alarm[mySeq].Time		:= 3000;

//Setup Sequence
step := D[900 + mySeq];
//Setup Pulse contact
pls := (step <> lastStep);
lastStep := step;

//Sequence
IF (step = 0) THEN
	//Disabled
END_IF;

//Bag Settled at buffer
ton_10ms_SettledBuffer(IN:= i_bagAtBuffer, PT:= bufferSettleTime);
IF (step = 1) THEN
	IF ton_10ms_SettledBuffer.Q AND NOT Std.HaltSysZone[myZone]THEN
		IF Line[myRelLine].Clear AND NOT i_bagAtBufferOut AND NOT i_bufferOutOpen AND NOT Line[myRelLine].Trip THEN
			IF (myBag = 0) THEN
				C[myRelLine] := 0;
				D[900 + mySeq] := 2;
			ELSIF (Bag[myBag].Cat > 0) AND (Bag[myOutBag].Cat = 0) THEN
				C[myRelLine] := 0;
				D[900 + mySeq] := 2;
			ELSIF (Bag[myBag].Cat = 0) THEN
				Alarm[mySeq].Name := ALM_BAG_DATA_ERROR;
				Alarm[mySeq].Time := 0;
			ELSIF (Bag[myOutBag].Cat > 0) THEN
				Alarm[mySeq].Name := ALM_BAG_DATA_ERROR;
				Alarm[mySeq].Bag := myOutBag;
				Alarm[mySeq].Time := 0;
			END_IF;
		ELSIF Line[myRelLine].Trip THEN
			Alarm[mySeq].Name := ALM_SWITCH_FAULT; //Trip is stuck on
			Alarm[mySeq].Time := 500;
		END_IF;
	ELSIF (myBag > 0) AND (Bag[myBag].Cat > 0) THEN
		Alarm[mySeq].Name := ALM_BAG_NOT_SETTLED;
	END_IF;
END_IF;

IF (step = 2) THEN
	dataValid := ((myBag = 0) OR ((Bag[myBag].Cat > 0) AND (Bag[myOutBag].Cat = 0)));
	o_openBuffer :=  dataValid;
	IF dataValid THEN
		IF Line[myRelLine].Trip THEN
			IF (myBag > 0) THEN
				Bag[myOutBag] := Bag[myBag];
				Bag[myBag]  := Bag[0];
			END_IF;
			D[900 + mySeq] := 1;
		END_IF;
		Alarm[mySeq].Name := ALM_BAG_NOT_RELEASED;
	ELSIF (myBag > 0) THEN
		IF (Bag[myBag].Cat = 0) THEN
			Alarm[mySeq].Name := ALM_BAG_DATA_ERROR;
			Alarm[mySeq].Time := 0;
		ELSIF (Bag[myOutBag].Cat > 0) THEN
			Alarm[mySeq].Name := ALM_BAG_DATA_ERROR;
			Alarm[mySeq].Bag := myOutBag;
			Alarm[mySeq].Time := 0;
		END_IF;
	END_IF;
END_IF;

//-----------------------------------
//PLC Outputs - adjust TO suit system
//-----------------------------------

Y[5].Y16 := o_openBuffer;

//Alarms
timerAlarm(IN := NOT pls AND (Alarm[mySeq].Name > 0),PT:= Alarm[mySeq].Time);

Alarm[mySeq].On 	:= timerAlarm.Q;
Alarm[mySeq].ET 	:= timerAlarm.ET;

END_PROGRAM
```

### Program Logical/Sequences/10ms/48_cp6 (IEC) - * SP2 Empty bags from SDC1/2

#### 12_sp2.var
```iecst
VAR RETAIN
	STEP : UINT;
	PLS : BOOL;
	LASTSTEP : UINT;
END_VAR
VAR
	TimerAlarm : TON_10ms;
	I_BagAtBuffer : ARRAY[0..3] OF BOOL;
	O_OpenBuffer : BOOL;
	SDC2BufferFullET : TIME;
	SDC2BufferFull : BOOL;
	SettledBufferET : TIME;
	SettledBuffer : ARRAY[0..3] OF BOOL;
	O_OpenSP2BufferStop : BOOL;
	O_SelectPoint : BOOL;
	SP2BufferFull : BOOL;
	SP2BufferFullET : UDINT;
	ParingLoopEnabled : BOOL;
	BagInLoopHasDest : BOOL;
	O_OpenSDC1BufferStop : BOOL;
	BagSettledAtBuffer : BOOL;
	BagSettledAtBufferET : UDINT;
	Alternator : USINT;
	I_OnLineA : BOOL;
	I_TiltA : BOOL;
	I_TiltB : BOOL;
	I_Bagout : BOOL;
	O_OpenBufferStop : BOOL;
	O_SelectLineA : BOOL;
	O_SelectLineB : BOOL;
	O_OpenStops : BOOL;
	O_TiltCylinder : BOOL;
	O_OperatePusher : BOOL;
	PointReset : BOOL;
	PointResetET : UDINT;
	BagAtTilt : BOOL;
	BagAtTiltET : UDINT;
	TiltDown : BOOL;
	TiltDownET : UDINT;
	TiltUp : BOOL;
	TiltUpET : UDINT;
	NotFull : BOOL;
	NotFullET : UDINT;
	Pushed : BOOL;
	SBSN1 : BOOL;
	SBSN1ET : UDINT;
	RequirePusherET : UDINT;
	PushedET : UDINT;
	I_BagAtBufferStop : BOOL;
	O_SP7ToSVC1 : BOOL;
	O_SP7ToSIC3 : BOOL;
	SDC1EmptyBufferFull : BOOL;
	SDC1EmptyBufferFullET : UDINT;
	Reset : BOOL;
	ResetET : UDINT;
	ResetPoint : BOOL;
	I_SDC1EmptyBagAtBuffer : BOOL;
	O_ResetPoints : BOOL;
	BagSettledSDC1Buffer : BOOL;
	BagSettledSDC1BufferET : UDINT;
	BagSettledSDC2Buffer : BOOL;
	BagSettledSDC2BufferET : UDINT;
	MySeq : USINT;
	BagSettledBufferET : ARRAY[0..3] OF UDINT;
	Alt : USINT;
	O_SelectCDC4 : BOOL;
	O_SelectStraight : BOOL;
	O_SelectCDC1 : BOOL;
	O_SelectCDC2 : BOOL;
END_VAR
```

#### 12_sp2Cyclic.ab
```automation-basic
PROGRAM _CYCLIC
	(* cyclic program *)

;---------------------------------------
;Sequence 12 - SP2 Single point 2 D[912]
;---------------------------------------

;Inputs

I_BagAtBuffer[1]		= X[5].X14
I_BagAtBuffer[2]		= X[5].X15

MySeq                   = 48

Alarm[MySeq].Name 			= 0
Alarm[MySeq].Bag			= 10001
Alarm[MySeq].Beacon		= TRUE
Alarm[MySeq].Extra			= 0
Alarm[MySeq].Time			= 3000

O_SelectCDC1                = FALSE
O_SelectCDC2             = FALSE

;Setup Sequence
STEP = D[900 + MySeq]
;Setup Pulse contact
PLS = (STEP <> LASTSTEP)
LASTSTEP = STEP

;Sequence
;Step 0 - Disabled
IF (STEP = 0) THEN
	;Disabled
ENDIF

;reset points
TON_10ms((STEP = 1),200,Reset,ResetET)
IF (STEP = 1) THEN

	IF (Line[47].Clear)  THEN
		D[900 + MySeq] = 2
	ENDIF
	ELSE

ENDIF

;check which bag is ready
TON_10ms(I_BagAtBuffer[1],200,SettledBuffer[1],BagSettledBufferET[1])
TON_10ms(I_BagAtBuffer[2],200,SettledBuffer[2],BagSettledBufferET[2])
IF (STEP = 2) THEN
	IF (Line[47].Clear) THEN
		Alt = Alt + 1
		IF (Alt > 2) THEN
			Alt = 0
		ENDIF
		IF SettledBuffer[1] AND (Alt = 1) THEN
			C[47]          = 0
		    D[900 + MySeq] = 3
		ELSE IF SettledBuffer[2] AND (Alt = 2) THEN
			C[47]          = 0
			D[900 + MySeq] = 4
		ENDIF
	ENDIF
ENDIF

;Bag at line
IF (STEP = 3) THEN
	O_SelectCDC1 = TRUE
	IF (Line[47].Trip = TRUE) THEN
		D[900 + MySeq] = 1
	ENDIF
	Alarm[MySeq].Name 	  = almBagNotArrived
ENDIF

;Bag at line
IF (STEP = 4) THEN
	O_SelectCDC2 = TRUE
	IF (Line[47].Trip = TRUE) THEN
		D[900 + MySeq] = 1
	ENDIF
	Alarm[MySeq].Name 	  = almBagNotArrived
ENDIF

;Alarms
TimerAlarm.IN 	= NOT PLS AND (Alarm[MySeq].Name > 0)
TimerAlarm.PT 	= Alarm[MySeq].Time
TimerAlarm FUB TON_10ms()
Alarm[MySeq].On 	= TimerAlarm.Q
Alarm[MySeq].ET 	= TimerAlarm.ET

;Outputs
Y[5].Y12 = O_SelectCDC1
Y[5].Y13 = O_SelectCDC2
END_PROGRAM
```

### Program Logical/Sequences/10ms/9_sic1_ref (IEC) - * SIC1 Incline Conveyor 1

#### 9_sic1Cyclic.ab
```automation-basic
PROGRAM _CYCLIC
	(* cyclic program *)

;---------------------------------------------------
;Sequence 12 - SIC1 Soiled Incline Conveyor 1 D[909]
;---------------------------------------------------

;Inputs

I_BagAtBuffer			= X[8].X06
I_PaddleInPosition		= X[6].X15
I_BagInIncline			= X[6].X14

O_OpenBufferStop		= FALSE
O_RunMotor 				= FALSE

I_BagAtOutgoingBuffer	= FALSE
O_OutgoingBufferOpen	= FALSE

Enable.IC[1]			= FALSE
O_SelectSDC1            = FALSE
O_SelectSDC2            = FALSE

Alarm[9].Name 			= 0
Alarm[9].Bag			= 287
Alarm[9].Beacon			= TRUE
Alarm[9].Extra			= 0
Alarm[9].Time			= 3000

;Setup Sequence
STEP = D[909]
;Setup Pulse contact
PLS = (STEP <> LASTSTEP)
LASTSTEP = STEP

;Sequence
;Step 0 - Disabled
IF (STEP = 0) THEN
	;Disabled
ENDIF

;Run Incline until paddle in position
IF (STEP = 1) THEN
	O_RunMotor = NOT I_PaddleInPosition
	IF I_PaddleInPosition THEN
		D[909] = 2
	ENDIF
	IF NOT Std.EStop THEN
		Alarm[9].Name = almSwitchFault
	ENDIF
ENDIF

;Wait for at buffer
TON_10ms(I_BagAtBuffer,300,BagAtBuffer,BagAtBufferET)
IF (STEP = 2) THEN
	IF (BagAtBuffer AND (Bag[240].Cat > 0) AND NOT Std.HaltSys) THEN
		D[909] = 3
	ENDIF
	IF (Bag[240].Cat > 0) AND NOT I_BagAtBuffer THEN
		Alarm[9].Name 	= almBagNotAtProx
		Alarm[9].Bag	= 240
	ELSE IF (Bag[240].Cat = 0) AND I_BagAtBuffer THEN
		Alarm[9].Name 	= almBagNotShownOnScreen
		Alarm[9].Bag	= 240
	ENDIF
ENDIF

;Open Buffer stop
IF (STEP = 3) THEN
	O_OpenBufferStop 	= TRUE
	Enable.IC[1]		= (NOT I_BagInIncline AND (Bag[240].Cat = 0))
	IF I_BagInIncline THEN
		D[909] = 4
	ENDIF
	;;Alarm[9].Name = almBagNotArrived
ENDIF

;Let bag settle at base of incline
TON_10ms((STEP = 4),300,BagSettled,BagSettledET)
IF (STEP = 4) THEN
	IF PLS AND (Bag[241].Cat = 0) AND (Bag[240].Cat > 0)  THEN
		Bag[241] = Bag[240]
		Bag[240] = Bag[0]
	ENDIF
	IF BagSettled THEN
		D[909] = 5
	ENDIF
ENDIF

;Move Bag up incline
TON_10ms((STEP = 5),800,BagNearTop,BagNearTopET)
IF (STEP = 5) THEN
	O_RunMotor = NOT BagNearTop
	IF BagNearTop THEN
		D[909] = 6
	ENDIF
	Alarm[9].Name = almSwitchFault
ENDIF

;Check for space at the ongoing buffer
;Run motor for 0.5 seconds
TON_10ms((STEP = 6),50,RunOn,RunOnET)
IF (STEP = 6) THEN
	O_RunMotor 		= NOT RunOn
	IF NOT Std.HaltSys THEN
		IF (Bag[242].Cat = 0) AND (Bag[241].Dst > 0) THEN
			Dest = Bag[241].Dst
			IF ((Dest = 21) AND Line[21].Clear AND (Bag[284].Cat = 0))THEN
				C[21]  = 0
				D[909] = 7
			ELSE IF ((Dest = 22) AND Line[22].Clear AND (Bag[273].Cat = 0))THEN
				C[22]  = 0
				D[909] = 8
			ENDIF

		ENDIF
	ENDIF
ENDIF

;Select SDCC 1 Buffer
IF (STEP = 7) THEN
	O_RunMotor 			= TRUE
	O_SelectSDC1        = TRUE

	IF ((Bag[241].Cat > 0) AND (Bag[242].Cat = 0)) THEN
		;Bag[241].Dst = 0
		Bag[242] = Bag[241]
		Bag[241] = Bag[0]
	ENDIF

	IF PLS THEN
		C[21] = 0
	ENDIF
	IF Line[21].Trip AND NOT PLS THEN
		IF ((Bag[242].Cat > 0) AND (Bag[284].Cat = 0)) THEN
			Bag[242].Dst = 0
			Bag[284] = Bag[242]
			Bag[242] = Bag[0]
		ENDIF
		D[909] = 1
	ENDIF
	;Alarm[9].Name = almBagNotReleased
ENDIF

;Select SDCC 1 Buffer
IF (STEP = 8) THEN
	O_RunMotor 			= TRUE
	O_SelectSDC2        = TRUE
	IF ((Bag[241].Cat > 0) AND (Bag[242].Cat = 0)) THEN
		;Bag[241].Dst = 0
		Bag[242] = Bag[241]
		Bag[241] = Bag[0]
	ENDIF

	IF PLS THEN
		C[22] = 0
	ENDIF
	IF (C[22] > 0) AND NOT PLS THEN
		IF ((Bag[242].Cat > 0) AND (Bag[274].Cat = 0)) THEN
			Bag[242].Dst = 0
			Bag[273] = Bag[242]
			Bag[242] = Bag[0]
		ENDIF
		D[909] = 1
	ENDIF
	;Alarm[9].Name = almBagNotReleased
ENDIF

;Alarms
TimerAlarm.IN 	= NOT PLS AND (Alarm[9].Name > 0)
TimerAlarm.PT 	= Alarm[9].Time
TimerAlarm FUB TON_10ms()
Alarm[9].On 	= TimerAlarm.Q
Alarm[9].ET 	= TimerAlarm.ET

;Outputs
Y[8].Y06 = O_OpenBufferStop
Y[2].Y09 = O_RunMotor
Y[8].Y14 = O_SelectSDC1
Y[8].Y15 = O_SelectSDC2
END_PROGRAM
```

### Program Logical/Sequences/10ms/0_sbelt (IEC) - * Loading and Sorting belts

#### 0_sbelt.var
```iecst
VAR
	I_SortBelt3Photo : BOOL;
	O_RunSortBelt1 : BOOL;
	O_RunSortBelt2 : BOOL;
	O_RunSortBelt3 : BOOL;
	SortBelt2RunningET : TIME;
	SortBelt3RunningET : TIME;
	O_RunSortBelt : ARRAY[0..7] OF BOOL;
END_VAR
```

#### 0_sbeltCyclic.ab
```automation-basic
PROGRAM _CYCLIC
(* cyclic program *)

;Inputs
	O_RunSortBelt[1]	= FALSE
	O_RunSortBelt[2]	= FALSE
	O_RunSortBelt[3]	= FALSE
	O_RunSortBelt[4]	= FALSE
	O_RunSortBelt[5]	= FALSE
	O_RunSortBelt[6]	= FALSE
	;Run belts
	O_RunSortBelt[1] =  NOT Std.EStop AND (NOT X[8].X13) AND (NOT Request.SB[2])
	O_RunSortBelt[2] =  NOT Std.EStop AND (NOT X[8].X13)
	O_RunSortBelt[3] =  NOT Std.EStop
	O_RunSortBelt[4] =  NOT Std.EStop
	O_RunSortBelt[5] =  NOT Std.EStop
	O_RunSortBelt[6] =  NOT Std.EStop

	;TON_10ms(O_RunSortBelt[3],300,O_RunSortBelt[2],SortBeltRunningET[2])
	;TON_10ms(O_RunSortBelt[2],300,O_RunSortBelt[1],SortBeltRunningET[1])

	;Outputs
	Y[14].Y03 = O_RunSortBelt[1]  AND (D[15]>0)
	Y[14].Y04 = O_RunSortBelt[2] AND (D[15]>0)
END_PROGRAM
```

### Program Logical/Sequences/10ms/50_stns1_7 (IEC) - *Sorting Stations--

#### stnsa.var
```iecst
VAR
	ContinuousSort : BOOL;
	TestStations : BOOL;
	Update : BOOL;
	LampTest : BOOL;
	I_PartLoad : ARRAY[0..50] OF BOOL;
	CloseFlap : ARRAY[0..50] OF BOOL;
	AllowRelease : ARRAY[0..50] OF BOOL;
END_VAR
VAR RETAIN
	BagOpened : ARRAY[0..50] OF BOOL;
	BagClosed : ARRAY[0..50] OF BOOL;
	OpenBag : ARRAY[0..50] OF BOOL;
END_VAR
VAR
	PLS : ARRAY[0..99] OF BOOL;
	AutoPurgeTrig : ARRAY[0..50] OF R_TRIG;
END_VAR
VAR RETAIN
	BagClosedET : ARRAY[0..50] OF TIME;
	BagOpenedET : ARRAY[0..50] OF TIME;
END_VAR
VAR
	TimerPartLoad : ARRAY[0..50] OF TON_10ms;
	TimerOpen : ARRAY[0..49] OF TON_10ms;
	TimerFlapClose : ARRAY[0..49] OF TON_10ms;
	TimerClosed : ARRAY[0..49] OF TON_10ms;
	TimerAlarm : ARRAY[0..49] OF TON_10ms;
	myBid : UDINT;
	StnBag : UINT;
	OpenTime : UINT;
	myBag : UINT;
	CloseTime : UINT;
END_VAR
VAR RETAIN
	STEP : UINT;
END_VAR
VAR
	mySeq : UINT;
	Bank : UINT;
END_VAR
VAR RETAIN
	n : UINT;
END_VAR
VAR
	myDisplayBag : UINT;
END_VAR
VAR RETAIN
	LASTSTEP : ARRAY[0..99] OF UINT;
END_VAR
VAR
	CloseFlapDelay : BOOL;
	CloseFlapDelayET : TIME;
	newBag : ARRAY[0..50] OF BOOL;
	myStnReg : UINT;
	myStnBit : UINT;
	testClose : BOOL;
	x : UINT;
END_VAR
```

#### stnsa.ab
```automation-basic
PROGRAM _CYCLIC
(* cyclic program *)

;Honeycombe Sorting Station Control
;----------------------------------------------------
;Revision 1.00 10/01/2002 D.J. First Issue
;Revision 2.00 07/02/2005 D.J. Removed Stn Mix
;Revision 3.00 22/08/2006 D.J. Changed to timer array
;----------------------------------------------------

mySeq = 50
Bank = 1

;Timers
OpenTime  = 700
CloseTime = 500

ContinuousSort = FALSE;(D[994] = 0)

;Lamp Test from TrackView
IF (BIT_TST(D[998],0) = 1) THEN
	LampTest = TRUE

ELSE
	LampTest = FALSE
ENDIF

	LOOP x = 1 TO Ldg[Bank].NoStations DO
		n = Ldg[Bank].Stations[x]

		;Parts Loads
		TimerPartLoad[n].IN		= I_PartLoad[n]
		TimerPartLoad[n].PT		= 100
		TimerPartLoad[n] FUB TON_10ms()

		IF TimerPartLoad[n].Q THEN
			D[800 + n] = 1
		ENDIF

		;Bag open timers
		TimerOpen[n].IN 		= OpenBag[n]
		TimerOpen[n].PT			= OpenTime
		TimerOpen[n] FUB TON_10ms()

		BagOpened[n] 			= TimerOpen[n].Q
		BagOpenedET[n]			= TimerOpen[n].ET

		;Bag closed timers
		TimerClosed[n].IN 		= NOT OpenBag[n]
		TimerClosed[n].PT		= CloseTime
		TimerClosed[n] FUB TON_10ms()

		BagClosed[n] 			= TimerClosed[n].Q
		BagClosedET[n]			= TimerClosed[n].ET

		;Update bag weight
		StnBag = LDG_GetBagFromStation(Std.StationBagsStart,n)
		Bag[StnBag].Wgt 		= Stn[n].Weight
		Bag[StnBag].Cnt 		= Stn[n].Count

		;Update Bag ID if cleared or zero
		IF ((BidStn > 0) AND (Bag[StnBag].Bid = 0) AND (Bag[StnBag].Cat > 0)) THEN
			Bag[StnBag].Bid = UINT(BidStn)
			BidStn			= 0
		ENDIF

		;Move bags from Display buffer position into Search array,,
		myDisplayBag = LDG_GetBagFromStation(Std.StationBagDisplay,n)

		;Keep Weight Live on Display
		Bag[myDisplayBag].Wgt = Stn[n].Weight
		Update = FALSE
		IF (Bag[StnBag].Cat <> Bag[myDisplayBag].Cat) THEN
			Update = TRUE
		ELSE IF (Bag[StnBag].Cus <> Bag[myDisplayBag].Cus) THEN
			Update = TRUE
		ELSE IF (Bag[StnBag].Prg <> Bag[myDisplayBag].Prg) THEN
			Update = TRUE
		ENDIF
		IF (Bag[myDisplayBag].Cat = Std.MaxCats) THEN
			Update = FALSE ; Do not update bag if Empty Bag is assigned.
			CloseFlap[n] = TRUE
		ELSE
			CloseFlap[n] = FALSE
		ENDIF

		;Flap close after above SP2 for 1 second
		TimerFlapClose[n].IN 	= Stn[n].SP2 AND (Bag[myDisplayBag].Cat <> Std.MaxCats)
		TimerFlapClose[n].PT	= 200 ;4 sec
		TimerFlapClose[n] FUB TON_10ms()

		IF ContinuousSort THEN
			AutoPurgeTrig[n].CLK = Update
			AutoPurgeTrig[n] FUB R_TRIG()
			IF AutoPurgeTrig[n].Q THEN
				newBag[n] = TRUE
			ENDIF

			IF (newBag[n] AND Std.AutoPurge AND NOT Stn[n].CloseFlap AND NOT Stn[n].ManualRelease AND NOT Stn[n].Purge AND NOT Stn[n].PurgeReverse)THEN
				D[800 + n] = 2 ; Bag change detected automatically purge the station... Weight is check in ZZstn
				newBag[n] = FALSE
			ENDIF

			IF ((NOT Stn[n].CloseFlap AND NOT Stn[n].ManualRelease AND NOT Stn[n].Purge AND NOT Stn[n].PurgeReverse AND (D[800 + n] = 0)) OR  (Bag[StnBag].Cat = 0)) THEN ;AND NOT Stn[n].SP2 THEN
				IF Update THEN;(Update AND (n <> 12)) THEN
					myBid = Bag[StnBag].Bid
					Bag[StnBag] = Bag[myDisplayBag]
					Bag[StnBag].Bid = myBid
				ENDIF
			ENDIF
		ELSE
			IF Update THEN
				myBid = Bag[StnBag].Bid
				Bag[StnBag] = Bag[myDisplayBag]
				Bag[StnBag].Bid = myBid
			ENDIF
		ENDIF

		;Ensure Display Bag has a  Bag ID
		IF ((BidStn > 0) AND (Bag[myDisplayBag].Bid = 0) AND  (Bag[myDisplayBag].Cat > 0)) THEN
			Bag[myDisplayBag].Bid = UINT(BidStn)
			BidStn			= 0
		ENDIF

		Alarm[mySeq + n].Name 		= 0
		Alarm[mySeq + n].Bag		= StnBag
		Alarm[mySeq + n].Beacon	= FALSE
		Alarm[mySeq + n].Extra		= 0
		Alarm[mySeq + n].Time		= 4000

		Stn[n].LampOn 		= FALSE
		Stn[n].GreenLamp	= FALSE

		STEP = D[900 + mySeq + n]
		;Setup Pulse contact
		PLS[n] = (STEP <> LASTSTEP[n])
		LASTSTEP[n] = STEP

		;Step 0 - Disabled
		IF (STEP = 0) THEN
			Stn[n].LampOn = TRUE
			Stn[n].CloseFlap = ((Bag[StnBag].Cat <> Bag[myDisplayBag].Cat))
			Stn[n].QTime = 0
			Stn[n].ManualRelease = 0
			Stn[n].Purge = 0
			;Disabled
		ENDIF

		IF (STEP = 1) THEN
			Stn[n].LampOn = TRUE
			Stn[n].GreenLamp = FALSE
			Stn[n].CloseFlap = TRUE
			myStnReg = (n > 32)
			IF (myStnReg = 0)THEN
				myStnBit =	n - 1
			ELSE IF (myStnReg = 1)THEN
				myStnBit = 	n - 33
			ELSE
				myStnBit = 0
			ENDIF
			Std.PurgeBank[Bank].StationsStatus[myStnReg] = BIT_CLR(Std.PurgeBank[Bank].StationsStatus[myStnReg],myStnBit)

	;		Stn[n].Purge = FALSE
	;		Stn[n].PurgeReverse = FALSE
			IF D[900 + 1] = n THEN
				D[900 + 1] = 0
			ENDIF
			IF BagClosed[n] THEN
				D[900 + mySeq + n] = 2
			ENDIF
			Alarm[mySeq + n].Name = almStationNotClosed
		ENDIF

		IF (STEP = 2) THEN
			Stn[n].LampOn = ((Stn[n].SP1 AND Std.Clock2s) OR Stn[n].SP2 OR (Stn[n].SP3 AND Std.Clock200ms))
			Stn[n].GreenLamp = ((NOT Stn[n].SP2 AND NOT Stn[n].SP3) OR TimerFlapClose[n].Q)
			;Close the flaps when the bag is above SP2
			IF TimerFlapClose[n].Q OR Stn[n].ManualRelease OR Stn[n].Purge OR Stn[n].PurgeReverse THEN
				Stn[n].CloseFlap 	= ContinuousSort
			ENDIF
			;Stop flap closing / re-open is bag below 3kg
			IF (Stn[n].Weight < 30) THEN
				Stn[n].CloseFlap 	= FALSE
			ENDIF
			IF ((D[900 + Std.StationBankReg + Bank] = n) AND Ldg[Bank].EnableStnRelease) THEN
				D[900 + mySeq + n] = 3
			ENDIF
			IF ((Bag[StnBag].Prg > 0) AND Stn[n].SP3) THEN
				Alarm[mySeq + n].Name = almBagOverWeight
			ENDIF
		ENDIF

		IF (STEP = 3) THEN
			Stn[n].LampOn = TRUE
			Stn[n].CloseFlap = ContinuousSort
			Stn[n].GreenLamp = TimerFlapClose[n].Q

			AllowRelease[n]  = TRUE

			IF (BagOpened[n] AND ((Stn[n].Weight < 30) OR Test.Stations) AND Ldg[Bank].BeltHasRun) THEN
				Stn[n].QTime 	= 0
				D[900 + mySeq + n] = 1
			ENDIF
			IF (Stn[n].Weight >= 30) THEN
				Alarm[mySeq + n].Name = almStationNotEmpty
			ENDIF
		ELSE
			AllowRelease[n]= FALSE
		ENDIF

		OpenBag[n] = AllowRelease[n];(STEP = 3)

		;Lamp Test
		IF LampTest THEN
			Stn[n].LampOn = TRUE
		ENDIF

		;Alarm timer
		TimerAlarm[n].IN 	= NOT PLS[n] AND (Alarm[mySeq + n].Name > 0)
		TimerAlarm[n].PT	= Alarm[mySeq + n].Time
		TimerAlarm[n] FUB TON_10ms()

		Alarm[mySeq + n].ET	= TimerAlarm[n].ET
		Alarm[mySeq + n].On 	= TimerAlarm[n].Q

;	Y[300 + n].Y07 = Stn[n].LampOn
;	Y[300 + n].Y05 = Stn[n].CloseFlap OR testClose
;	Y[300 + n].Y06 = Stn[n].GreenLamp
;	Y[300 + n].Y04 = OpenBag[n]

ENDLOOP

;Outputs
;-------
;	YG05 = OpenBag[1]
;	YG06 = OpenBag[2]
;	YG07 = OpenBag[3]
;	YG08 = OpenBag[4]
;	YH05 = OpenBag[5]
;	YH06 = OpenBag[6]
;	YH07 = OpenBag[7]
;	YH08 = OpenBag[8]
;	YJ05 = OpenBag[9]
;	YJ06 = OpenBag[10]
;	YJ07 = OpenBag[11]
;	YJ08 = OpenBag[12]
;	YK05 = OpenBag[13]
;	YK06 = OpenBag[14]
;	YK07 = OpenBag[15]
;	YK08 = OpenBag[16]

	Y[12].Y05 = OpenBag[1] ;ok
	Y[12].Y06 = OpenBag[2]
	Y[12].Y07 = OpenBag[3]
	Y[12].Y08 = OpenBag[4]

	Y[13].Y05 = OpenBag[5];ok
	Y[13].Y06 = OpenBag[6]
	Y[13].Y07 = OpenBag[7]
;	Y[32].Y08 = OpenBag[8]

;	Y[33].Y05 = OpenBag[9]
;	Y[33].Y06 = OpenBag[10]
;	Y[33].Y07 = OpenBag[11]
;	Y[33].Y08 = OpenBag[12]

;	Y[34].Y05 = OpenBag[13]
;	Y[34].Y06 = OpenBag[14]
;	Y[34].Y07 = OpenBag[15]
;	Y[34].Y08 = OpenBag[16]

	Y[12].Y01 = Stn[1].LampOn ;ok
	Y[12].Y02 = Stn[2].LampOn
	Y[12].Y03 = Stn[3].LampOn
	Y[12].Y04 = Stn[4].LampOn

	Y[13].Y01 = Stn[5].LampOn ;ok
	Y[13].Y02 = Stn[6].LampOn
	Y[13].Y03 = Stn[7].LampOn
;	Y[32].Y04 = Stn[8].LampOn

;	Y[33].Y01 = Stn[9].LampOn
;	Y[33].Y02 = Stn[10].LampOn
;	Y[33].Y03 = Stn[11].LampOn
;	Y[33].Y04 = Stn[12].LampOn

;	Y[34].Y01 = Stn[13].LampOn
;	Y[34].Y02 = Stn[14].LampOn
;	Y[34].Y03 = Stn[15].LampOn
;	Y[34].Y04 = Stn[16].LampOn

END_PROGRAM
```

### Program Logical/Sequences/10ms/50_stn8_14 (IEC) - *Sorting Stations--

#### stnsa.ab
```automation-basic
PROGRAM _CYCLIC
(* cyclic program *)

;Honeycombe Sorting Station Control
;----------------------------------------------------
;Revision 1.00 10/01/2002 D.J. First Issue
;Revision 2.00 07/02/2005 D.J. Removed Stn Mix
;Revision 3.00 22/08/2006 D.J. Changed to timer array
;----------------------------------------------------

mySeq = 50
Bank = 2

;Timers
OpenTime  = 700
CloseTime = 500

ContinuousSort = FALSE;(D[994] = 0)

;Lamp Test from TrackView
IF (BIT_TST(D[998],0) = 1) THEN
	LampTest = TRUE

ELSE
	LampTest = FALSE
ENDIF

	LOOP x = 8 TO Ldg[Bank].NoStations DO
;	LOOP x = 12 TO 12 DO
		n = Ldg[Bank].Stations[x]

		;Parts Loads
		TimerPartLoad[n].IN		= I_PartLoad[n]
		TimerPartLoad[n].PT		= 100
		TimerPartLoad[n] FUB TON_10ms()

		IF TimerPartLoad[n].Q THEN
			D[800 + n] = 1
		ENDIF

		;Bag open timers
		TimerOpen[n].IN 		= OpenBag[n]
		TimerOpen[n].PT			= OpenTime
		TimerOpen[n] FUB TON_10ms()

		BagOpened[n] 			= TimerOpen[n].Q
		BagOpenedET[n]			= TimerOpen[n].ET

		;Bag closed timers
		TimerClosed[n].IN 		= NOT OpenBag[n]
		TimerClosed[n].PT		= CloseTime
		TimerClosed[n] FUB TON_10ms()

		BagClosed[n] 			= TimerClosed[n].Q
		BagClosedET[n]			= TimerClosed[n].ET

		;Update bag weight
		StnBag = LDG_GetBagFromStation(Std.StationBagsStart,n)
		Bag[StnBag].Wgt 		= Stn[n].Weight
		Bag[StnBag].Cnt 		= Stn[n].Count

		;Update Bag ID if cleared or zero
		IF ((BidStn > 0) AND (Bag[StnBag].Bid = 0) AND (Bag[StnBag].Cat > 0)) THEN
			Bag[StnBag].Bid = UINT(BidStn)
			BidStn			= 0
		ENDIF

		;Move bags from Display buffer position into Search array,,
		myDisplayBag = LDG_GetBagFromStation(Std.StationBagDisplay,n)

		;Keep Weight Live on Display
		Bag[myDisplayBag].Wgt = Stn[n].Weight
		Update = FALSE
		IF (Bag[StnBag].Cat <> Bag[myDisplayBag].Cat) THEN
			Update = TRUE
		ELSE IF (Bag[StnBag].Cus <> Bag[myDisplayBag].Cus) THEN
			Update = TRUE
		ELSE IF (Bag[StnBag].Prg <> Bag[myDisplayBag].Prg) THEN
			Update = TRUE
		ENDIF
		IF (Bag[myDisplayBag].Cat = Std.MaxCats) THEN
			Update = FALSE ; Do not update bag if Empty Bag is assigned.
			CloseFlap[n] = TRUE
		ELSE
			CloseFlap[n] = FALSE
		ENDIF

		;Flap close after above SP2 for 1 second
		TimerFlapClose[n].IN 	= Stn[n].SP2 AND (Bag[myDisplayBag].Cat <> Std.MaxCats)
		TimerFlapClose[n].PT	= 200 ;4 sec
		TimerFlapClose[n] FUB TON_10ms()

		IF ContinuousSort THEN
			AutoPurgeTrig[n].CLK = Update
			AutoPurgeTrig[n] FUB R_TRIG()
			IF AutoPurgeTrig[n].Q THEN
				newBag[n] = TRUE
			ENDIF

			IF (newBag[n] AND Std.AutoPurge AND NOT Stn[n].CloseFlap AND NOT Stn[n].ManualRelease AND NOT Stn[n].Purge AND NOT Stn[n].PurgeReverse)THEN
				D[800 + n] = 2 ; Bag change detected automatically purge the station... Weight is check in ZZstn
				newBag[n] = FALSE
			ENDIF

			IF ((NOT Stn[n].CloseFlap AND NOT Stn[n].ManualRelease AND NOT Stn[n].Purge AND NOT Stn[n].PurgeReverse AND (D[800 + n] = 0)) OR  (Bag[StnBag].Cat = 0)) THEN ;AND NOT Stn[n].SP2 THEN
				IF Update THEN;(Update AND (n <> 12)) THEN
					myBid = Bag[StnBag].Bid
					Bag[StnBag] = Bag[myDisplayBag]
					Bag[StnBag].Bid = myBid
				ENDIF
			ENDIF
		ELSE
			IF Update THEN
				myBid = Bag[StnBag].Bid
				Bag[StnBag] = Bag[myDisplayBag]
				Bag[StnBag].Bid = myBid
			ENDIF
		ENDIF

		;Ensure Display Bag has a  Bag ID
		IF ((BidStn > 0) AND (Bag[myDisplayBag].Bid = 0) AND  (Bag[myDisplayBag].Cat > 0)) THEN
			Bag[myDisplayBag].Bid = UINT(BidStn)
			BidStn			= 0
		ENDIF

		Alarm[mySeq + n].Name 		= 0
		Alarm[mySeq + n].Bag		= StnBag
		Alarm[mySeq + n].Beacon	= FALSE
		Alarm[mySeq + n].Extra		= 0
		Alarm[mySeq + n].Time		= 4000

		Stn[n].LampOn 		= FALSE
		Stn[n].GreenLamp	= FALSE

		STEP = D[900 + mySeq + n]
		;Setup Pulse contact
		PLS[n] = (STEP <> LASTSTEP[n])
		LASTSTEP[n] = STEP

		;Step 0 - Disabled
		IF (STEP = 0) THEN
			Stn[n].LampOn = TRUE
			Stn[n].CloseFlap = ((Bag[StnBag].Cat <> Bag[myDisplayBag].Cat))
			Stn[n].QTime = 0
			Stn[n].ManualRelease = 0
			Stn[n].Purge = 0
			;Disabled
		ENDIF

		IF (STEP = 1) THEN
			Stn[n].LampOn = TRUE
			Stn[n].GreenLamp = FALSE
			Stn[n].CloseFlap = TRUE
			myStnReg = (n > 32)
			IF (myStnReg = 0)THEN
				myStnBit =	n - 1
			ELSE IF (myStnReg = 1)THEN
				myStnBit = 	n - 33
			ELSE
				myStnBit = 0
			ENDIF
			Std.PurgeBank[Bank].StationsStatus[myStnReg] = BIT_CLR(Std.PurgeBank[Bank].StationsStatus[myStnReg],myStnBit)

	;		Stn[n].Purge = FALSE
	;		Stn[n].PurgeReverse = FALSE
			IF D[950] = n THEN
				D[950] = 0
			ENDIF
			IF BagClosed[n] THEN
				D[900 + mySeq + n] = 2
			ENDIF
			Alarm[mySeq + n].Name = almStationNotClosed
		ENDIF

		IF (STEP = 2) THEN
			Stn[n].LampOn = ((Stn[n].SP1 AND Std.Clock2s) OR Stn[n].SP2 OR (Stn[n].SP3 AND Std.Clock200ms))
			Stn[n].GreenLamp = ((NOT Stn[n].SP2 AND NOT Stn[n].SP3) OR TimerFlapClose[n].Q)
			;Close the flaps when the bag is above SP2
			IF TimerFlapClose[n].Q OR Stn[n].ManualRelease OR Stn[n].Purge OR Stn[n].PurgeReverse THEN
				Stn[n].CloseFlap 	= ContinuousSort
			ENDIF
			;Stop flap closing / re-open is bag below 3kg
			IF (Stn[n].Weight < 30) THEN
				Stn[n].CloseFlap 	= FALSE
			ENDIF
			IF ((D[900 + 50] = n) AND Ldg[Bank].EnableStnRelease) THEN
				D[900 + mySeq + n] = 3
			ENDIF
			IF ((Bag[StnBag].Prg > 0) AND Stn[n].SP3) THEN
				Alarm[mySeq + n].Name = almBagOverWeight
			ENDIF
		ENDIF

		IF (STEP = 3) THEN
			Stn[n].LampOn = TRUE
			Stn[n].CloseFlap = ContinuousSort
			Stn[n].GreenLamp = TimerFlapClose[n].Q

			AllowRelease[n]  = TRUE

			IF (BagOpened[n] AND ((Stn[n].Weight < 30) OR Test.Stations) AND Ldg[Bank].BeltHasRun) THEN
				Stn[n].QTime 	= 0
				D[900 + mySeq + n] = 1
			ENDIF
			IF (Stn[n].Weight >= 30) THEN
				Alarm[mySeq + n].Name = almStationNotEmpty
			ENDIF
		ELSE
			AllowRelease[n]= FALSE
		ENDIF

		OpenBag[n] = AllowRelease[n];(STEP = 3)

		;Lamp Test
		IF LampTest THEN
			Stn[n].LampOn = TRUE
		ENDIF

		;Alarm timer
		TimerAlarm[n].IN 	= NOT PLS[n] AND (Alarm[mySeq + n].Name > 0)
		TimerAlarm[n].PT	= Alarm[mySeq + n].Time
		TimerAlarm[n] FUB TON_10ms()

		Alarm[mySeq + n].ET	= TimerAlarm[n].ET
		Alarm[mySeq + n].On 	= TimerAlarm[n].Q

;	Y[300 + n].Y07 = Stn[n].LampOn
;	Y[300 + n].Y05 = Stn[n].CloseFlap OR testClose
;	Y[300 + n].Y06 = Stn[n].GreenLamp
;	Y[300 + n].Y04 = OpenBag[n]

ENDLOOP

;Outputs
;-------
;	YG05 = OpenBag[1]
;	YG06 = OpenBag[2]
;	YG07 = OpenBag[3]
;	YG08 = OpenBag[4]
;	YH05 = OpenBag[5]
;	YH06 = OpenBag[6]
;	YH07 = OpenBag[7]
;	YH08 = OpenBag[8]
;	YJ05 = OpenBag[9]
;	YJ06 = OpenBag[10]
;	YJ07 = OpenBag[11]
;	YJ08 = OpenBag[12]
;	YK05 = OpenBag[13]
;	YK06 = OpenBag[14]
;	YK07 = OpenBag[15]
;	YK08 = OpenBag[16]

;	Y[31].Y05 = OpenBag[1] ;ok
;	Y[31].Y06 = OpenBag[2]
;	Y[31].Y07 = OpenBag[3]
;	Y[31].Y08 = OpenBag[4]

;	Y[32].Y05 = OpenBag[5];ok
;	Y[32].Y06 = OpenBag[6]
;	Y[32].Y07 = OpenBag[7]
	Y[14].Y05 = OpenBag[8]

	Y[14].Y06 = OpenBag[9]
	Y[14].Y07 = OpenBag[10]
	Y[14].Y08 = OpenBag[11]
	Y[15].Y05 = OpenBag[12]

	Y[15].Y06 = OpenBag[13]
	Y[15].Y07 = OpenBag[14]
;	Y[15].Y07 = OpenBag[15]
;	Y[34].Y08 = OpenBag[16]

;	Y[31].Y01 = Stn[1].LampOn ;ok
;	Y[31].Y02 = Stn[2].LampOn
;	Y[31].Y03 = Stn[3].LampOn
;	Y[31].Y04 = Stn[4].LampOn

;	Y[32].Y01 = Stn[5].LampOn ;ok
;	Y[32].Y02 = Stn[6].LampOn
;	Y[32].Y03 = Stn[7].LampOn
	Y[14].Y01 = Stn[8].LampOn

	Y[14].Y02 = Stn[9].LampOn
	Y[14].Y03 = Stn[10].LampOn
	Y[14].Y04 = Stn[11].LampOn
	Y[15].Y01 = Stn[12].LampOn

	Y[15].Y02 = Stn[13].LampOn
	Y[15].Y03 = Stn[14].LampOn
;	Y[34].Y03 = Stn[15].LampOn
;	Y[34].Y04 = Stn[16].LampOn

END_PROGRAM
```

### Program Logical/Sequences/10ms/2_svc3 (IEC) - * SVC1 Up from SLU1 & Loading

#### 8_svc1.var
```iecst
VAR RETAIN
	I_CarrAtTop : BOOL;
	I_CarrAtBottom : BOOL;
	STEP : UINT;
	PLS : BOOL;
	LASTSTEP : UINT;
	O_MoveCarrUp : BOOL;
	O_OpenCarrStop : BOOL;
	O_MoveCarrDown : BOOL;
	I_BagOnCarr : BOOL;
END_VAR
VAR
	O_OpenBuffer : BOOL;
	BagSettledOnCarr : BOOL;
	BagSettledOnCarrET : TIME;
	I_BagReleased : BOOL;
	TimerAlarm : TON_10ms;
	I_CarrAtMiddle : BOOL;
	I_CarrAtWeighing : BOOL;
	I_NoEmptyBag : BOOL;
	I_CollectEmpty : BOOL;
	I_UseAsLoading : BOOL;
	I_UpPushButton : BOOL;
	I_DownPushButton : BOOL;
	Dst : UINT;
	PButton : BOOL;
	SVCRaw : DINT;
	n : UINT;
	ValidCus : BOOL;
	ValidWgt : BOOL;
	O_AlarmLamp : BOOL;
	ValidCat : BOOL;
	Choice : ARRAY[0..4] OF UINT;
	PButtonET : TIME;
	Status : UINT;
	PastMiddleET : TIME;
	PastMiddle : BOOL;
	ValidDst : BOOL;
	I_CarrAtEmtyBagIn : BOOL;
	I_CarrAtEmptyBagOut : BOOL;
	I_FullBagReleased : BOOL;
	I_EmptyBagReleased : BOOL;
	I_FullBagAtBuffer : BOOL;
	I_WeighBeamOverRide : BOOL;
	O_MoveCarrDownToBottom : BOOL;
	O_MoveCarrDownToEmptyIn : BOOL;
	O_MoveCarrDownToEmptyBagOut : BOOL;
	OpenBufferStop : BOOL;
	NoEmptyBag : BOOL;
	BagSettledAtStop : BOOL;
	weighbeambag : INT;
	OverWeight : BOOL;
	OVERLOAD : UINT;
	LowWeight : UINT;
	UnderWeight : BOOL;
	BagSettledAtStopET : UDINT;
	WeightOK : BOOL;
	WeightOKET : UDINT;
END_VAR
```

#### 8_svc1Cyclic.ab
```automation-basic
PROGRAM _CYCLIC
	(* cyclic program *)

;--------------------------------------------
;Sequence 8 - SVC1 Vertical conveyor 1 D[908]
;--------------------------------------------

;Inputs
I_CarrAtTop				= X[3].X01
I_CarrAtBottom			= X[3].X02
I_CarrAtEmtyBagIn       = X[3].X03
I_CarrAtEmptyBagOut     = X[3].X04
I_BagOnCarr				= X[3].X05
I_FullBagReleased	    = X[3].X07
I_EmptyBagReleased	    = X[8].X06

I_FullBagAtBuffer		= X[3].X06
I_WeighBeamOverRide     = X[5].X12

O_OpenBuffer				= FALSE
O_MoveCarrUp				= FALSE
O_MoveCarrDownToBottom		= FALSE
O_MoveCarrDownToEmptyIn 	= FALSE
O_MoveCarrDownToEmptyBagOut = FALSE
O_OpenCarrStop				= FALSE
OpenBufferStop              = FALSE

Request.SVCEmptyBag[1]		= FALSE ;request to SP7
Request.SVCFullBag[1]       = FALSE ;request to SVC2

Alarm[8].Name 			= 0
Alarm[8].Bag			= 294
Alarm[8].Beacon			= FALSE
Alarm[8].Extra			= 0
Alarm[8].Time			= 3000

;Setup Sequence
STEP = D[908]
;Setup Pulse contact
PLS = (STEP <> LASTSTEP)
LASTSTEP = STEP

;Sequence
IF (STEP = 0) THEN
	;Disabled
ENDIF

;Move carriage down to Empty IN
IF (STEP = 1) THEN
	O_MoveCarrDownToEmptyIn = NOT I_CarrAtEmtyBagIn
	IF I_CarrAtEmtyBagIn THEN
		D[908] = 2
	ENDIF
	IF NOT Std.EStop THEN
		Alarm[8].Name = almCarriageMoveFault
	ENDIF
ENDIF

;Check Status
IF (STEP = 2) THEN
	IF (NOT I_BagOnCarr AND (Bag[294].Cat = 0) AND NOT I_CarrAtTop) THEN
		D[908] = 3
	ENDIF
	IF (Bag[294].Cat > 0) THEN
		Alarm[8].Name = almBagDataError
	ELSE IF I_BagOnCarr OR I_CarrAtTop THEN
		Alarm[8].Name = almSwitchFault
	ENDIF
ENDIF

;Check opreation mode
IF (STEP = 3) THEN
	Request.SVCEmptyBag[1] = TRUE ;request bto SP7

	IF Enable.SVCEmptyBag[1] AND NOT Std.HaltSys THEN
		D[908] = 4
	ENDIF
	IF (NoEmptyBag AND BagSettledAtStop AND (C[30] = 2)) THEN
		D[908] = 9  ;if no bag at buffer and full bag at buffer below then go and get
	ENDIF
ENDIF

;wait for bag to arrive from SP7
IF (STEP = 4) THEN
	Request.SVCEmptyBag[1] = TRUE
	IF I_BagOnCarr THEN
		D[908] = 5
	ENDIF
	Alarm[8].Name = almBagNotArrived
ENDIF

;Let bag settle on carriage
TON_10ms(I_BagOnCarr,20,BagSettledOnCarr,BagSettledOnCarrET)
IF (STEP = 5) THEN

	IF BagSettledOnCarr THEN
		D[908] = 6
	ENDIF
	Alarm[8].Name = almBagNotSettled
ENDIF

;Move Carriage down to empty out position
IF (STEP = 6) THEN
	O_MoveCarrDownToEmptyBagOut = NOT I_CarrAtEmptyBagOut
	IF I_CarrAtEmptyBagOut THEN
		D[908] = 7
	ENDIF
	IF NOT Std.EStop THEN
		Alarm[8].Name = almCarriageMoveFault
	ENDIF
ENDIF

;Check if buffer is clear
IF (STEP = 7) THEN
	IF NOT Std.HaltSys THEN
		IF NOT Y[8].Y06 AND NOT I_EmptyBagReleased AND Line[29].Clear THEN ;check low level empty buffer is clear
			D[908] = 8
		ENDIF
	ENDIF
	;IF I_BagReleased THEN
	;Alarm[8].Name = almSwitchFault
	;ENDIF
ENDIF

;Open carriage stop let empty bag out
IF (STEP = 8) THEN
	O_OpenCarrStop = I_CarrAtEmptyBagOut
	IF PLS THEN
		C[29] 	= 0
	ENDIF

	IF (PLS AND (D[903] = 1)) THEN
		D[903] = 2
	ENDIF

	IF I_EmptyBagReleased THEN
		D[908] 	= 9
	ENDIF
	IF NOT Std.EStop THEN
		Alarm[8].Name = almBagNotReleased
	ENDIF
ENDIF

;Check Middle position switch
IF (STEP = 9) THEN
	IF (NOT I_FullBagAtBuffer AND (Bag[292].Cat = 0) AND NOT I_BagOnCarr) THEN
		D[908] = 19
	ENDIF

	IF NOT I_CarrAtBottom THEN
		D[908] = 10
	ENDIF
	Alarm[8].Name = almSwitchFault
ENDIF

;move down to full bag in
IF (STEP = 10) THEN
	O_MoveCarrDownToBottom = NOT I_CarrAtBottom
	IF  I_CarrAtBottom THEN
		D[908] = 11
	ENDIF
	Alarm[8].Name = almSwitchFault
ENDIF

;Calculate weight
AI351RAW_02
SVCRaw = DINT(AI351RAW_01)
SVCRaw = (SVCRaw * 1000) ;2000
IF (SVCRaw > 0) THEN
	weighbeambag = INT(SVCRaw / 32767)
ELSE
	weighbeambag = 0
ENDIF
IF (Bag[292].Cat > 0) AND (D32[120] <>Bag[292].Cat ) THEN
			D32[120] := Bag[292].Cat
ENDIF

;Over Weight
IF ((weighbeambag > D32[125]) AND NOT I_WeighBeamOverRide AND (STEP = 11)) THEN
	OverWeight = TRUE
	D[81] = 1
ELSE
	OverWeight = FALSE
	D[81] = 0
ENDIF

Bag[370].Cat = 1
Bag[370].Wgt = weighbeambag

OVERLOAD = uint(D32[125]);Over weight SP3
LowWeight= uint(D32[123]) ;SP1

UnderWeight = (weighbeambag <(D32[123]));Under weight

;Full Bag at buffer stop
TON_10ms(I_FullBagAtBuffer AND (Bag[292].Cat > 0),300,BagSettledAtStop,BagSettledAtStopET)
IF (STEP = 11) THEN
	TON_10ms(NOT OverWeight,100,WeightOK,WeightOKET)
	IF BagSettledAtStop AND NOT I_BagOnCarr  THEN
		IF (weighbeambag <(D32[123])) AND WeightOK OR I_WeighBeamOverRide THEN
			IF UnderWeight THEN
				ReportLoading[17].Cat = UINT(Bag[292].Cat)	;Category
					ReportLoading[17].Cus = Bag[292].Cus			;Customer
					ReportLoading[17].Wgt = UINT(Bag[370].Wgt)		;Weight
					ReportLoading[17].Cnt = 17						;Count
					ReportLoading[17].Stn = 17        				;Station
					ReportLoading[17].Mcn = 17						;Machine
			ENDIF
			D[908] = 12
		ELSE IF UnderWeight THEN
			Alarm[8].Time = 10
			Alarm[8].Bag				= 292
			Alarm[8].Name = almBagDataError
			;D[82] = 1

		ELSE
			Alarm[8].Time = 10
			Alarm[8].Bag				= 292
			;Alarm[8].Name = almBagOverWeight
			;D[82] = 0
		ENDIF

	ENDIF

	IF I_BagOnCarr THEN
		Alarm[8].Name = almSwitchFault
	ELSE IF OverWeight THEN
		Alarm[8].Time = 10
		Alarm[8].Bag				= 292
		Alarm[8].Name = almBagOverWeight
	ENDIF
ENDIF

;Open buffer stop
IF (STEP = 12) THEN
	OpenBufferStop = I_CarrAtBottom
	IF ((Bag[292].Cat > 0) AND (Bag[293].Cat = 0)) THEN
		Bag[293] = Bag[292]
		Bag[292] = Bag[0]
	ENDIF

	IF I_BagOnCarr THEN
		Bag[294] = Bag[293]
		Bag[293] = Bag[0]
		D[908] = 13
	ENDIF
	IF NOT Std.EStop THEN
		Alarm[8].Name = almBagNotReleased
	ENDIF
ENDIF

;Bag settles on carriage
IF (STEP = 13) THEN
	IF BagSettledOnCarr THEN
		D[908] = 14
	ENDIF
ENDIF

;check status
IF (STEP = 14) THEN
	IF NOT I_CarrAtTop THEN
		D[908] = 15
	ENDIF
ENDIF

;move carriage up
IF STEP = 15 THEN
	O_MoveCarrUp = NOT I_CarrAtTop
	IF I_CarrAtTop AND NOT Enable.SVCFullBag[1] THEN
		D[908] = 16
	ENDIF
ENDIF

;request a bag to SVC2
IF (STEP = 16) THEN

		Request.SVCFullBag[1] = TRUE
	IF (Enable.SVCFullBag[1] AND NOT I_FullBagReleased AND (Bag[295].Cat = 0)) THEN
		C[14]  = 0
		D[908] = 17
	ENDIF
ENDIF

;open carriage stop
IF (STEP = 17) THEN
	O_OpenCarrStop = I_CarrAtTop
	IF PLS THEN
		C[14] = 0
	ENDIF

	IF ((Bag[294].Cat > 0) AND (Bag[295].Cat = 0)) THEN
		Bag[295] = Bag[294]
		Bag[294] = Bag[0]
	ENDIF

	IF Line[14].Clear AND NOT PLS THEN
		D[908] = 18
	ENDIF
ENDIF

;Check status
IF STEP = 18 THEN
	IF NOT I_CarrAtEmtyBagIn THEN
		D[908] = 1
	ENDIF
ENDIF

;Go to top
IF STEP = 19 THEN
	O_MoveCarrUp = NOT I_CarrAtTop
	IF I_CarrAtTop THEN
		D[908] = 1
	ENDIF
ENDIF

;Alarms
TimerAlarm.IN 	= NOT PLS AND (Alarm[8].Name > 0)
TimerAlarm.PT 	= Alarm[8].Time
TimerAlarm FUB TON_10ms()
Alarm[8].On 	= TimerAlarm.Q
Alarm[8].ET 	= TimerAlarm.ET

;PLC Outputs
;-----------
Y[12].Y01 		= (O_MoveCarrUp 	AND NOT I_CarrAtTop)
Y[12].Y02 		= (O_MoveCarrDownToEmptyIn OR O_MoveCarrDownToBottom  OR O_MoveCarrDownToEmptyBagOut)
;Y[12].Y03 		= O_MoveCarrDownToEmptyBagOut

Y[12].Y04 		= O_OpenCarrStop
Y[3].Y06        = OpenBufferStop

;Don't allow forcing of carriage movement and carriage stop
YForceDisable[12].Y01 = TRUE
YForceDisable[12].Y02 = TRUE
YForceDisable[12].Y04 = TRUE
YForceDisable[12].Y05 = TRUE

END_PROGRAM
```

### Program Logical/Sequences/10ms/5_spf1 (IEC) - * Soiled Offgoing Transfer Lines 1 - 14

#### 5_spf1.var
```iecst
VAR RETAIN
	STEP : UINT;
	LASTSTEP : UINT;
	PLS : BOOL;
	BagSettledTime : ARRAY[0..99] OF UINT;
	Destination : UINT;
	SettleTime : UINT;
	BestTime : UINT;
	LineSelect : ARRAY[0..49] OF BOOL;
	ResetPointsET : TIME;
	ResetPoints : BOOL;
	n : UINT;
	IncSettle : BOOL;
	LineSettle : ARRAY[0..99] OF BOOL;
	I_BagAtStop : ARRAY[0..49] OF BOOL;
	OffGoingEnable : BOOL;
	AlarmBagNotProx : BOOL;
	SearchDest : UINT;
END_VAR
VAR
	TimerAlarm : TON_10ms;
	MaxBuffers : UINT;
	ResetBrush : BOOL;
	FoundLine : UINT;
	O_Reset : BOOL;
	O_SDCBufferOpen : ARRAY[0..4] OF BOOL;
	I_SDCBagAtBuffer : ARRAY[0..4] OF BOOL;
	ResetBrushET : TIME;
	SVC2BufferClear : BOOL;
	CloseBrush : BOOL;
	SDC4_Valid : BOOL;
	I_BagPassedSVC2 : BOOL;
	EnableSDC3Search : BOOL;
	EnableSDC1Search : BOOL;
	Alternator : UINT;
	LastDest : UINT;
	I_ApproachBrush : BOOL;
	O_CloseBrush : BOOL;
	SDC1_Valid : BOOL;
	SDC2_Valid : BOOL;
	SDC3_Valid : BOOL;
	EmptyInTransit : BOOL;
	CloseStop : BOOL;
	I_BagReleased : BOOL;
	BufferBag : ARRAY[0..4] OF UINT;
	BufferClear : ARRAY[0..4] OF BOOL;
	testAtStop : BOOL;
	PairingLoop : BOOL;
END_VAR
```

### Program Logical/Sequences/10ms/9_svc2 (IEC, version 1.00.0) - * SVC2 Vertical Conveyor

#### 17_svc2Cyclic.ab
```automation-basic
PROGRAM _CYCLIC
	(* cyclic program *)

;--------------------------------------------
;Sequence 7 - SVC1 Vertical conveyor 1 D[907]
;--------------------------------------------

mySeq                   = 9

;Inputs
I_CarrAtTop				= X[3].X09
I_CarrAtBottom			= X[3].X10
I_CarrAtEmptyBagIn      = X[3].X11
I_CarriageAtEmptyBagOut = X[3].X12

I_BagOnCarr				= X[3].X13
I_BagAtEmptyBuffer		= X[3].X14 ;bag at buffer stop H\L
I_BagAtFullBuffer       = X[3].X15 ;bag at full buffer low level

I_EmptyBagAtBufferStop  = X[9].X06 ;bag at low level buffer stop low level
I_FullBagAtBufferStop   = X[7].X16 ;bag at H\L buffer stop full bag

O_EmptyBagAtBufferStop  = Y[9].Y06 ;empty buffer stop low level
O_FullBagAtBufferStop   = Y[7].Y16 ;full bag buffer stop H\L

O_OpenEmptyBufferStop	= FALSE ;Y314
O_OpenFullBufferStop    = FALSE ;Y315

O_MoveCarrUp			= FALSE
O_MoveCarrDown			= FALSE
O_MoveCarrDown1         = FALSE
O_MoveCarrDown2         = FALSE
O_OpenCarrStop			= FALSE
Alarm[mySeq].Name 		= 0
Alarm[mySeq].Bag		= 225
Alarm[mySeq].Beacon		= TRUE
Alarm[mySeq].Extra		= 0
Alarm[mySeq].Time		= 6000

;Setup Sequence
STEP = D[900 + mySeq]
;Setup Pulse contact
PLS = (STEP <> LASTSTEP)
LASTSTEP = STEP

;Safety switch check
IF ((STEP = 1) OR (STEP = 5) OR (STEP = 10)) THEN
	IF I_Disable THEN
		D[900 + mySeq] = 0
	ENDIF
ENDIF

;Sequence
IF (STEP = 0) THEN
	;Disabled
ENDIF

;Move carriage down to empty bag in
TON_10ms((STEP = 1),100,StopClosed,StopClosedET)
IF (STEP = 1) THEN
	O_MoveCarrDown = (NOT I_CarrAtEmptyBagIn AND NOT I_CarrAtBottom)
	IF (I_CarrAtEmptyBagIn  = TRUE) THEN
		D[909] = 2
	ENDIF
	IF NOT Std.EStop THEN
		Alarm[mySeq].Name = ALM_CARRIAGE_MOVE_FAULT
	ENDIF
ENDIF

;empty bag at buffer stop
TON_10ms(I_BagAtEmptyBuffer,200,BagSettledAtBuffer,BagSettledAtBufferET)
IF (STEP = 2) THEN
	IF (NOT I_BagOnCarr AND (BagSettledAtBuffer = TRUE)) THEN
		D[909] = 3
	;ELSE IF ((D[16] = 0) AND BagAtBuffer AND (E[1950] > 0)) THEN
	    ;D[909] = 15 ; TAKE OUT
	ENDIF
ENDIF

;open buffer stop
IF (STEP = 3) THEN
	O_OpenEmptyBufferStop = I_CarrAtEmptyBagIn
	IF I_BagOnCarr THEN
		D[909] = 4
	ENDIF
ENDIF

;bag settles on carriage
TON_10ms(I_BagOnCarr,300,BagSettledOnCarr,BagSettledOnCarrET)
IF (STEP = 4) THEN
	IF BagSettledOnCarr THEN
		D[909] = 5
	ENDIF
	Alarm[mySeq].Time		= 1600
	Alarm[mySeq].Name = ALM_BAG_NOT_SETTLED
ENDIF

;move carriage down
IF (STEP = 5) THEN
	O_MoveCarrDown1 	= NOT I_CarriageAtEmptyBagOut ;down to empty bag out
	IF I_CarriageAtEmptyBagOut THEN
		D[909] = 6
	ENDIF
	IF NOT Std.EStop THEN
		Alarm[mySeq].Time		= 1000
		Alarm[mySeq].Name = ALM_CARRIAGE_MOVE_FAULT
	ENDIF
ENDIF

;check buffer clear
TON_10ms((NOT I_EmptyBagAtBufferStop AND NOT O_EmptyBagAtBufferStop),300,BufferClear,BufferClearET)
             ;X906                             ;Y906
IF (STEP = 6) THEN

	IF (Line[32].Clear AND (BufferClear = TRUE))THEN
		C[32] = 0
		D[909] = 7
	ENDIF
ENDIF

;Open carr stop
IF (STEP = 7) THEN
	O_OpenCarrStop = I_CarriageAtEmptyBagOut
	D[48]          = 4

	IF ((C[32] >=1) AND (I_EmptyBagAtBufferStop = TRUE) AND NOT I_CarrAtBottom) THEN
		D[909] = 8
	ENDIF
	Alarm[mySeq].Time		= 600
	Alarm[mySeq].Name = ALM_BAG_NOT_RELEASED
ENDIF

;move carriage down to bottom
IF (STEP = 8) THEN
	O_MoveCarrDown2 = NOT I_CarrAtBottom
	IF I_CarrAtBottom THEN
		D[909] = 9
	ENDIF
	IF NOT Std.EStop THEN
		Alarm[mySeq].Time		= 1000
		Alarm[mySeq].Name = ALM_CARRIAGE_MOVE_FAULT
	ENDIF
ENDIF

;Wait for full bag
TON_10ms(I_BagAtFullBuffer,300,BagAtBuffer,BagAtBufferET)
;TON_10ms(NoBag,2000,GetEmptyBag,GetEmptyBagET)
IF (STEP = 9) THEN
	IF BagAtBuffer AND (Bag[222].Cat > 0) AND NOT I_BagOnCarr THEN
		D[909] = 10
	ENDIF
;	NoBag = (NOT BagAtBuffer AND (E[1950] = 0) AND (E[1930] = 0) AND Line[34].Clear)
;	IF GetEmptyBag THEN
		;D[909] = 15
;	ENDIF
ENDIF

;Open carr stop
IF (STEP = 10) THEN
	O_OpenFullBufferStop = I_CarrAtBottom
	IF I_BagOnCarr THEN
		D[909] = 11
	ENDIF
ENDIF

;Bag settles on carr
IF (STEP = 11) THEN
	IF (Bag[222].Cat>0) AND (Bag[225].Cat = 0) THEN
		Bag[225] = Bag[222]
		Bag[222] = Bag[0]
	ENDIF
	IF BagSettledOnCarr THEN
		D[909] = 12
	ENDIF
	Alarm[mySeq].Time		= 1600
	Alarm[mySeq].Name = almBagNotSettled
ENDIF

;Send carriage up
IF (STEP = 12) THEN
	O_MoveCarrUp = NOT I_CarrAtTop
	IF I_CarrAtTop THEN
		D[909] = 13
	ENDIF
	IF NOT Std.EStop THEN
		Alarm[mySeq].Time		= 1000
		Alarm[mySeq].Name = ALM_CARRIAGE_MOVE_FAULT
	ENDIF
ENDIF

;check buffer clear and stop not open,bag at stop input not made
IF (STEP = 13) THEN
	IF ((Line[20].Clear = TRUE) AND NOT O_FullBagAtBufferStop AND NOT I_FullBagAtBufferStop) THEN
		C[20]  = 0
		D[909] = 14
	ENDIF
ENDIF

;Wait for bag out hoist

IF (STEP = 14) THEN
	IF PLS THEN
		C[20] = 0
	ENDIF
	O_OpenCarrStop = I_CarrAtTop
	IF ((Line[20].Full = TRUE) AND (I_FullBagAtBufferStop = TRUE)AND NOT PLS) THEN
		IF (Bag[225].Cat>0) AND (Bag[227].Cat = 0) THEN
		Bag[227] = Bag[225]
		Bag[225] = Bag[0]
	ENDIF
		D[909] = 1
	ENDIF
	Alarm[mySeq].Time		= 1000
	Alarm[mySeq].Name = ALM_BAG_NOT_RELEASED
ENDIF
;Alarms
TimerAlarm.IN 	= NOT PLS AND (Alarm[mySeq].Name > 0)
TimerAlarm.PT 	= Alarm[mySeq].Time
TimerAlarm FUB TON_10ms()
Alarm[mySeq].On 	= TimerAlarm.Q
Alarm[mySeq].ET 	= TimerAlarm.ET

;PLC Outputs
;-----------
Y[3].Y14 = O_OpenEmptyBufferStop
Y[3].Y15 = O_OpenFullBufferStop

Y[13].Y06 = (O_MoveCarrUp 	AND NOT I_CarrAtTop)
Y[13].Y07 =  O_MoveCarrDown

Y[13].Y08 = O_MoveCarrDown1
Y[13].Y09 = O_MoveCarrDown2

Y[13].Y10 = O_OpenCarrStop
Y[3].Y15 = O_OpenFullBufferStop

;Don't allow forcing of carriage movement and carriage stop
YForceDisable[13].Y06 	= TRUE
YForceDisable[13].Y07	= TRUE
YForceDisable[13].Y08 	= TRUE
END_PROGRAM
```

#### 17_svc2.var
```iecst
VAR RETAIN
	STEP : UINT;
	PLS : BOOL;
	LASTSTEP : UINT;
	O_OpenBufferStop : BOOL;
	I_BagAtBuffer : BOOL;
	O_RunMotor : BOOL;
	BagSettled : BOOL;
	BagSettledET : TIME;
	BagAtBuffer : BOOL;
	RunOnET : TIME;
	RunOn : BOOL;
	BagNearTopET : TIME;
	BagNearTop : BOOL;
	BagAtBufferET : UDINT;
	I_BagInIncline : BOOL;
END_VAR
VAR
	I_BagAtOutgoingBuffer : BOOL;
	I_PaddleInPosition : BOOL;
	CloseBufferStop : BOOL;
	CloseBufferStopET : TIME;
	O_OutgoingBufferOpen : BOOL;
	TimerAlarm : TON_10ms;
	O_SelectSP4ToSP2 : BOOL;
	I_BagReleased : BOOL;
	O_SelectSP4 : BOOL;
	I_BagOutAtTop : BOOL;
	I_BagOutAtBottom : BOOL;
	I_BagOnCarriage : BOOL;
	I_CarriageAtTop : BOOL;
	I_CarriageAtBottom : BOOL;
	O_OpenCarriageStop : BOOL;
	O_MoveUp : BOOL;
	O_MoveDown : BOOL;
	I_BagAtSVCBuffer : BOOL;
	O_BufferStop : BOOL;
	Carrstoptimer : BOOL;
	CarrstoptimerET : TIME;
	I_BagOutAtTopSVC2 : BOOL;
	I_BagOnCarriageSVC2 : BOOL;
	I_CarrAtTop : BOOL;
	I_CarrAtBottom : BOOL;
	I_CarrAtFullIn : BOOL;
	I_BagOnCarr : BOOL;
	O_OpenBuffer : BOOL;
	O_MoveCarrUp : BOOL;
	O_MoveCarrDown : BOOL;
	O_OpenCarrStop : BOOL;
	O_SelectSP1 : BOOL;
	O_SelectSP8 : BOOL;
	BagSettledOnCarr : BOOL;
	BagSettledOnCarrET : UDINT;
	PairedBagSVC2 : BOOL;
	LoopPairDest : BOOL;
	PairOnLoop : BOOL;
	BagPassed : BOOL;
	BagPassedET : UDINT;
	TRUEO_BufferStop : BOOL;
	mySeq : INT;
	myReportStn : INT;
	I_CarriageAtEmptyIn : BOOL;
	I_EmptyBagAtBuffer : BOOL;
	I_LoadingSequence : BOOL;
	I_UnloadingSequence : BOOL;
	I_UpButton : BOOL;
	O_MoveRailIn : BOOL;
	O_MoveRailOut : BOOL;
	O_IndicatorLamp : BOOL;
	O_SVC1PanelLamp : BOOL;
	SVC1AtWeight : BOOL;
	SVC1Amber : BOOL;
	FlashAmberLamp : BOOL;
	I_Disable : BOOL;
	FlashAmberLampET : UDINT;
	SVC1AtWeightET : UDINT;
	SVC2ValidWeight : BOOL;
	Pushbutton : BOOL;
	PushbuttonET : UDINT;
	WeightFault : BOOL;
	WeightFaultET : UDINT;
	SVC2_OK : BOOL;
	SVC1ValidWeight : BOOL;
	SVC1Alarm : BOOL;
	n : USINT;
	LineSearch : ARRAY[0..5] OF UINT;
	Choice : INT;
	LineValid : BOOL;
	SVC2Alarm : INT;
	SafeStop : BOOL;
	BagSettledAtBuffer : BOOL;
	BagSettledAtBufferET : UDINT;
	BagSettledOnCarriage : BOOL;
	BagSettledOnCarriageET : UDINT;
	SVC2AtWeight : BOOL;
	TimeDelay : BOOL;
	TimeDelayET : UDINT;
	I_CarrAtEmptyBagIn : BOOL;
	I_CarriageAtEmptyBagOut : BOOL;
	I_BagAtEmptyBuffer : BOOL;
	I_BagAtFullBuffer : BOOL;
	I_EmptyBagAtBufferStop : BOOL;
	I_FullBagAtBufferStop : BOOL;
	O_EmptyBagAtBufferStop : BOOL;
	O_FullBagAtBufferStop : BOOL;
	O_OpenEmptyBufferStop : BOOL;
	O_OpenFullBufferStop : BOOL;
	O_MoveCarrDown1 : BOOL;
	O_MoveCarrDown2 : BOOL;
	StopClosed : BOOL;
	StopClosedET : UDINT;
	BufferClear : BOOL;
	BufferClearET : UDINT;
END_VAR
```

### Program Logical/Sequences/10ms/10_svc3 (IEC) - * SVC3 Vertical Conveyor

#### 18_svc3.var
```iecst
VAR RETAIN
	STEP : UINT;
	PLS : BOOL;
	LASTSTEP : UINT;
	O_OpenBufferStop : BOOL;
	I_BagAtBuffer : BOOL;
	O_RunMotor : BOOL;
	BagSettled : BOOL;
	BagSettledET : TIME;
	BagAtBuffer : BOOL;
	RunOnET : TIME;
	RunOn : BOOL;
	BagNearTopET : TIME;
	BagNearTop : BOOL;
	BagAtBufferET : UDINT;
	I_BagInIncline : BOOL;
END_VAR
VAR
	I_BagAtOutgoingBuffer : BOOL;
	zzTON_10ms00002 : TON_10ms;
	zzTON_10ms00003 : TON_10ms;
	I_PaddleInPosition : BOOL;
	zzTON_10ms00004 : TON_10ms;
	CloseBufferStop : BOOL;
	CloseBufferStopET : TIME;
	O_OutgoingBufferOpen : BOOL;
	TimerAlarm : TON_10ms;
	O_SelectSP4ToSP2 : BOOL;
	I_BagReleased : BOOL;
	O_SelectSP4 : BOOL;
	I_BagOutAtTop : BOOL;
	I_BagOutAtBottom : BOOL;
	I_BagOnCarriage : BOOL;
	I_CarriageAtTop : BOOL;
	I_CarriageAtBottom : BOOL;
	O_OpenCarriageStop : BOOL;
	O_MoveUp : BOOL;
	O_MoveDown : BOOL;
	I_BagAtBufferStop : BOOL;
	BagSettledAtBuffer : BOOL;
	BagSettledAtBufferET : TIME;
	BufferClear : BOOL;
	I_BagOutAtTopSVC3 : BOOL;
	I_CarrAtTop : BOOL;
	I_CarrAtBottom : BOOL;
	I_CarrAtFullBagIn : BOOL;
	I_BagOnCarr : BOOL;
	O_SP1Bend : BOOL;
	O_SP3Straight : BOOL;
	O_SP8Bend : BOOL;
	O_OpenBuffer : BOOL;
	O_MoveCarrUp : BOOL;
	O_MoveCarrDown : BOOL;
	O_OpenCarrStop : BOOL;
	O_SP3Bend : BOOL;
	SettledBuffer : BOOL;
	SettledBufferET : UDINT;
	ParingLoopEnabled : BOOL;
	BagSettledOnCarr : BOOL;
	BagSettledOnCarrET : UDINT;
	PairOnLoop : BOOL;
	PairNotValidSVC3 : BOOL;
	HLBagMatch : BOOL;
	NoPairForSVC3 : BOOL;
	LLBagMatch : BOOL;
	CarriagePasted : BOOL;
	CarriagePastedET : UDINT;
	mySeq : INT;
	O_BufferStop : BOOL;
END_VAR
```

#### 18_svc3Cyclic.ab
```automation-basic
PROGRAM _CYCLIC
	(* cyclic program *)

;---------------------------------------------------
;Sequence 13 - SIC2 Soiled Incline Conveyor 2 D[913]
;---------------------------------------------------
mySeq                   = 10
;Inputs
I_CarrAtTop				= X[10].X01
I_CarrAtBottom			= X[10].X02

I_BagAtBuffer           = X[10].X05
I_BagOnCarr				= X[10].X03

O_MoveCarrUp			= FALSE
O_MoveCarrDown			= FALSE

O_OpenCarrStop			= FALSE
O_BufferStop            = FALSE

Request.VC[3]          = FALSE

Alarm[10].Name 			= 0
Alarm[10].Bag			= 231
Alarm[10].Beacon		= TRUE
Alarm[10].Extra			= 0
Alarm[10].Time			= 3000
;Setup Sequence
STEP = D[910]
;Setup Pulse contact
PLS = (STEP <> LASTSTEP)
LASTSTEP = STEP

;Sequence
;Step 0 - Disabled
IF (STEP = 0) THEN
	IF I_BagOnCarr	THEN
		Alarm[10].Time			= 3
		Alarm[mySeq].Name = ALM_SWITCH_FAULT
	ENDIF
ENDIF

;Move carriage down to bottom
IF (STEP = 1) THEN
	O_MoveCarrDown = TRUE
	IF (I_CarrAtBottom  = TRUE) THEN
		D[910] = 2
	ENDIF
	IF NOT Std.EStop THEN
		Alarm[10].Time			= 1000
		Alarm[mySeq].Name = ALM_CARRIAGE_MOVE_FAULT
	ENDIF
	IF I_BagOnCarr	THEN
		Alarm[10].Time			= 3
		Alarm[mySeq].Name = ALM_SWITCH_FAULT
		D[910] = 0
	ENDIF
ENDIF

;bag at buffer stop
TON_10ms(I_BagAtBuffer,300,BagSettledAtBuffer,BagSettledAtBufferET)
IF (STEP = 2) THEN
	IF (BagSettledAtBuffer AND (Bag[230].Cat > 0) AND NOT I_BagOnCarr) THEN
		D[910] = 3
	ENDIF
ENDIF

;open buffer stop
IF (STEP = 3) THEN
	O_BufferStop = TRUE
	IF I_BagOnCarr THEN
		D[910] = 4
	ENDIF
	Alarm[10].Time			= 900
	Alarm[mySeq].Name = almBagNotArrived
ENDIF

;bag settles on carriage
TON_10ms(I_BagOnCarr,300,BagSettledOnCarr,BagSettledOnCarrET)
IF (STEP = 4) THEN
	IF (Bag[230].Cat>0) AND (Bag[231].Cat = 0) THEN
		Bag[231] = Bag[230]
		Bag[230] = Bag[0]
	ENDIF
	IF (BagSettledOnCarr = TRUE) THEN
		D[910] = 5
	ENDIF
	Alarm[mySeq].Time		= 1600
	Alarm[mySeq].Name = almBagNotSettled
ENDIF

;move carriage up
IF (STEP = 5) THEN
	O_MoveCarrUp 	= TRUE
								  ;enable from SP3 off    trans bag
	IF ((I_CarrAtTop = TRUE) AND NOT Enable.VC[3] AND (Bag[232].Cat = 0)) THEN

		D[910] = 6
	ENDIF
	IF NOT Std.EStop THEN
		Alarm[mySeq].Time		= 1000
		Alarm[mySeq].Name = ALM_CARRIAGE_MOVE_FAULT
	ENDIF
ENDIF

;check SP3 is clear
IF (STEP = 6) THEN
	Request.VC[3] = TRUE
	IF Enable.VC[3] THEN
		C[36]  = 0
		D[910] = 7
	ENDIF
ENDIF

;Open carr stop
IF (STEP = 7) THEN
	IF PLS THEN
		C[36] =0
	ENDIF
	O_OpenCarrStop = I_CarrAtTop
	IF (Bag[231].Cat>0) AND (Bag[232].Cat = 0) THEN
		Bag[232] = Bag[231]
		Bag[231] = Bag[0]
	ENDIF

	IF ((Line[36].Clear = TRUE) AND NOT PLS) THEN
		D[910] = 1
	ENDIF
	Alarm[mySeq].Time		= 600
	Alarm[mySeq].Name = ALM_BAG_NOT_RELEASED

ENDIF

;Alarms
TimerAlarm.IN 	= NOT PLS AND (Alarm[10].Name > 0)
TimerAlarm.PT 	= Alarm[10].Time
TimerAlarm FUB TON_10ms()
Alarm[10].On 	= TimerAlarm.Q
Alarm[10].ET 	= TimerAlarm.ET

;PLC Outputs
;-----------
;Outputs
Y[13].Y11 = (O_MoveCarrUp AND NOT I_CarrAtTop)
Y[13].Y12 = (O_MoveCarrDown AND NOT I_CarrAtBottom)
Y[10].Y05 = (O_BufferStop AND  I_CarrAtBottom)

Y[13].Y13 = (O_OpenCarrStop AND I_CarrAtTop)

;Don't allow forcing of carriage movement and carriage stop
YForceDisable[13].Y11 = TRUE
YForceDisable[13].Y12 = TRUE

END_PROGRAM
```

### Program Logical/Sequences/10ms/13_bson (IEC, version 1.00.0) - * SBSN1 Bagstacker Ongoing 

#### 14_bsonCyclic.ab
```automation-basic
PROGRAM _CYCLIC
(* cyclic program *)

;----------------------------------------
;Sequence 14 - Ongoing Bag Stacker D[914]
;----------------------------------------

;Inputs
I_BagAtBuffer			= FALSE ;X[7].X01
I_OnLineA		  		= X[7].X01
I_TiltA					= X[7].X02
I_TiltB					= X[7].X03
I_Bagout				= X[7].X04

O_OpenBufferStop		= FALSE
O_SelectLineA			= FALSE
O_SelectLineB			= FALSE
O_OpenStops				= FALSE
O_TiltCylinder			= FALSE
O_OperatePusher			= FALSE

Request.BSN[1]			= FALSE

Alarm[13].Name 			= 0
Alarm[13].Bag			= 10014
Alarm[13].Beacon		= FALSE
Alarm[13].Extra			= 0
Alarm[13].Time			= 3000

;Setup Sequence
STEP = D[913]
;Setup Pulse contact
PLS = (STEP <> LASTSTEP)
LASTSTEP = STEP

;Sequence
IF (STEP = 0) THEN
	;Disabled
ENDIF

;Select Line 'A'
TON_10ms((STEP = 1),100,PointReset,PointResetET)
IF (STEP = 1) THEN
	;O_SelectLineA = NOT PointReset
	SwtichesOk = (NOT I_OnLineA AND NOT I_TiltA AND NOT I_TiltB)
	IF SwtichesOk AND PointReset AND NOT Std.HaltSys THEN
		D[913] = 2
	ENDIF
	IF NOT SwtichesOk THEN
		Alarm[13].Name = almSwitchFault
	ENDIF
ENDIF

;Wait for bag at buffer
TON_10ms(I_BagAtBuffer,300,BagAtBuffer,BagAtBufferET)
IF (STEP = 2) THEN
	Request.BSN[1] = TRUE
	IF (Enable.BSN[1] = TRUE) THEN
		D[913] = 3
	ENDIF
ENDIF

;Open buffer stop
IF (STEP = 3) THEN
O_SelectLineA  = TRUE
	Request.BSN[1] = TRUE
	IF I_OnLineA THEN
		D[913] = 4
	ENDIF
	Alarm[13].Name = almBagNotArrived
ENDIF

;Select Line 'B' and Wait for bag in Tilt position
TON_10ms((I_TiltA AND I_TiltB),300,BagAtTilt,BagAtTiltET)
IF (STEP = 4) THEN
	Request.BSN[1] = TRUE
	O_SelectLineB = TRUE
	IF BagAtTilt THEN
		D[913] = 5
	ENDIF
	Alarm[13].Name = almBagNotSettled
ENDIF

;Tilt down
TON_10ms((STEP = 5),500,TiltDown,TiltDownET)
TON_10ms(TiltDown,200,Pusher,PusherET)
IF (STEP = 5) THEN
	O_TiltCylinder = TRUE
	O_Pusher       = TiltDown and not Pusher
	IF TiltDown AND Pusher THEN
		D[913] = 6
	ENDIF
ENDIF

;Tilt up
TON_10ms((STEP = 6),500,TiltUp,TiltUpET)
IF (STEP = 6) THEN
	IF TiltUp THEN
		D[913] = 7
	ENDIF
ENDIF

;Check not full
TON_10ms(NOT I_Bagout,300,NotFull,NotFullET)
IF (STEP = 7) THEN
	IF NotFull THEN
		D[913] = 8
	ENDIF
ENDIF

;Open stops to release bag
IF (STEP = 8) THEN
	O_OpenStops = TRUE
	IF I_Bagout THEN
		D[913] = 1
	ENDIF
	Alarm[13].Name = almBagNotReleased
ENDIF

;Pusher Cylinder
TON_10ms((STEP = 8) AND NOT Pushed,500,O_OperatePusher,RequirePusherET)
TON_10ms(O_OperatePusher,500,Pushed,PushedET)

;Alarms
TimerAlarm.IN 	= NOT PLS AND (Alarm[13].Name > 0)
TimerAlarm.PT 	= Alarm[13].Time
TimerAlarm FUB TON_10ms()
Alarm[13].On 	= TimerAlarm.Q
Alarm[13].ET 	= TimerAlarm.ET

;Outputs
Y[7].Y06 = O_Pusher
Y[7].Y01 = O_SelectLineA
Y[7].Y02 = O_SelectLineB
Y[7].Y04 = O_TiltCylinder
Y[7].Y03 = O_OpenStops
Y[7].Y05 = O_OperatePusher
END_PROGRAM
```

### Program Logical/Sequences/10ms/14_bsoff (IEC, version 1.00.0) - * SBSF1 Bagstacker Offgoing

#### 15_bsoffCyclic.ab
```automation-basic
PROGRAM _CYCLIC
  	(* cyclic program *)

;-----------------------------------------
;Sequence 15 - Offgoing Bag Stacker D[915]
;-----------------------------------------

;Inputs
I_RockSepA				= X[7].X07
I_RockSepB				= X[7].X08
I_TiltA					= X[7].X09
I_TiltB					= X[7].X10
I_OutLineA				= X[7].X11
I_OutLineB				= X[7].X12

O_OpenRockSep			= FALSE
O_LevelCylinder			= FALSE
O_OpenLineAStop			= FALSE
O_OpenLineBStop			= FALSE
O_SelectLineA			= FALSE
O_SelectLineB			= FALSE

Alarm[14].Name 			= 0
Alarm[14].Bag			= 10002
Alarm[14].Beacon		= FALSE
Alarm[14].Extra			= 0
Alarm[14].Time			= 3000

;Setup Sequecne
STEP = D[914]
;Setup Pulse contact
PLS = (STEP <> LASTSTEP)
LASTSTEP = STEP

;Sequence

;Select Line 'A'
TON_10ms((NOT I_TiltA AND NOT I_TiltB),100,LevelClear,LevelClearET)
IF (STEP = 1) THEN
	IF LevelClear AND NOT Std.HaltSys THEN
		D[914] = 2
	ENDIF
	IF NOT Std.HaltSys THEN
		Alarm[14].Name = almSwitchFault
	ENDIF
ENDIF

;Open seperators wait for leveller to be ready
TON_10ms(((STEP = 2) AND I_RockSepA AND I_RockSepB),200,SettledInSeps,SettledInSepsET)
IF (STEP = 2) THEN
	O_OpenRockSep = TRUE
	IF SettledInSeps THEN
		D[914] = 3
	ENDIF
	;Alarm[15].Name = almBagNotArrived
ENDIF

;Wait for bag to settle in leveller position
TON_10ms((I_TiltA AND I_TiltB),300,SettledLevel,SettledLevelET)
IF (STEP = 3) THEN
	IF SettledLevel THEN
		D[914] = 4
	ENDIF
	Alarm[14].Name = almBagNotSettled
ENDIF

;Move bag leveller down
TON_10ms((STEP = 4),500,LevellerDown,LevellerDownET)
IF (STEP = 4) THEN
	O_LevelCylinder = TRUE
	IF LevellerDown THEN
		D[914] = 5
	ENDIF
ENDIF

;Allow bag leveller to retract
TON_10ms((STEP = 5),500,LevellerUp,LevellerUpET)
IF (STEP = 5) THEN
	O_LevelCylinderUP = TRUE
	IF LevellerUp THEN
		D[914] = 6
	ENDIF
ENDIF

;Check room in Buffer
EmptyBufferStopClear = NOT X[8].X08 AND NOT Y[8].Y08
IF (STEP = 6) THEN
	IF NOT Std.HaltSys THEN
		IF (Line[35].Clear AND EmptyBufferStopClear) THEN
			C[35]  = 0
			D[914] = 7
		ENDIF
	ENDIF
ENDIF

;Open stop on line 'A'
IF (STEP = 7) THEN
	O_OpenLineAStop = TRUE
	O_SelectLineA 	= TRUE
	;IF PLS THEN
	;	C[17] = 0
	;ENDIF
	IF I_OutLineA THEN
		D[914] = 8
	ENDIF
	Alarm[14].Name = almBagNotReleased
ENDIF

;Open stop on line 'B'
IF (STEP = 8) THEN
	O_OpenLineBStop = TRUE
	O_SelectLineA 	= TRUE
	IF I_OutLineB THEN
		D[914] = 9
	ENDIF
	Alarm[14].Name = almBagNotReleased
ENDIF

;Select bag stop and wait for bag out of leveller
IF (STEP = 9) THEN
	O_SelectLineB = TRUE
	IF Line[35].Trip THEN
		D[914] = 1
	ENDIF
	Alarm[14].Name = almBagNotReleased
ENDIF

;Alarms
TimerAlarm.IN 	= NOT PLS AND (Alarm[14].Name > 0)
TimerAlarm.PT 	= Alarm[14].Time
TimerAlarm FUB TON_10ms()
Alarm[14].On 	= TimerAlarm.Q
Alarm[14].ET 	= TimerAlarm.ET

;Outputs
Y[7].Y08 = O_OpenRockSep
Y[7].Y11 = O_LevelCylinder
Y[7].Y09 = O_OpenLineAStop
Y[7].Y10 = O_OpenLineBStop
Y[7].Y12 = O_SelectLineA
Y[7].Y13 = O_SelectLineB

;SPR1 Offgoing Bagstacker Pressure relief
TON_10ms((NOT X[10].X07 AND NOT X[10].X08),500,Y[10].Y07,PRLineClearET[0])

;SPR2 Offgoing Bagstacker Pressure relief
TON_10ms((NOT X[10].X09 AND NOT X[10].X10),500,Y[10].Y09,PRLineClearET[1])

;SPR3 Offgoing Bagstacker Pressure relief
TON_10ms((NOT X[10].X11 AND NOT X[10].X12),500,Y[10].Y11,PRLineClearET[2])
;TON_10ms((NOT X[7].X05 AND NOT X[7].X06),500,Y[7].Y07,PRLineClearET[4])
;TON_10ms((NOT X[7].X05 AND X[7].X05),500,Y[7].Y07,PRLineClearET[3])
TON_10ms((NOT X[7].X05 AND NOT X[7].X06),500,Openseparator,OpenseparatorET)

Y[7].Y07 = Openseparator

END_PROGRAM
```

#### 15_bsoff.var
```iecst
VAR RETAIN
	STEP : UINT;
	PLS : BOOL;
	LASTSTEP : UINT;
	LevellerDownET : TIME;
	O_LevelCylinder : BOOL;
	O_SelectLineB : BOOL;
	O_SelectLineA : BOOL;
	I_OutLineB : BOOL;
	LevellerDown : BOOL;
	LevellerUp : BOOL;
	LevellerUpET : TIME;
	I_TiltB : BOOL; (* SPR1 Trolley past stop *)
	I_OutLineA : BOOL;
	O_OpenRockSep : BOOL;
	O_OpenLineAStop : BOOL;
	O_OpenLineBStop : BOOL;
	I_RockSepA : BOOL;
	I_RockSepB : BOOL;
	I_TiltA : BOOL; (* SBS1 ON Bag on stacker *)
	O_LevelCylinderUP : BOOL;
END_VAR
VAR
	PRLineClearET : ARRAY[0..4] OF TIME;
	SettledLevel : BOOL;
	SettledLevelET : TIME;
	SettledInSepsET : TIME;
	SettledInSeps : BOOL;
	LevelClearET : TIME;
	LevelClear : BOOL;
	TimerAlarm : TON_10ms;
	EmptyBufferStopClear : BOOL;
	Openseparator : BOOL;
	OpenseparatorET : UDINT;
END_VAR
```

### Program Logical/Sequences/10ms/15_spXX (IEC) - * SP2 Empty bags from SDC1/2

#### 12_sp2.var
```iecst
VAR RETAIN
	STEP : UINT;
	PLS : BOOL;
	LASTSTEP : UINT;
END_VAR
VAR
	TimerAlarm : TON_10ms;
	I_BagAtBuffer : BOOL;
	O_OpenBuffer : BOOL;
	SDC2BufferFullET : TIME;
	SDC2BufferFull : BOOL;
	SettledBufferET : TIME;
	SettledBuffer : BOOL;
	O_OpenSP2BufferStop : BOOL;
	O_SelectPoint : BOOL;
	SP2BufferFull : BOOL;
	SP2BufferFullET : UDINT;
	ParingLoopEnabled : BOOL;
	BagInLoopHasDest : BOOL;
	O_OpenSDC1BufferStop : BOOL;
	BagSettledAtBuffer : BOOL;
	BagSettledAtBufferET : UDINT;
	Alternator : USINT;
	O_SP5Straight : BOOL;
	O_SP5Bend : BOOL;
	I_BagAtBufferStop : BOOL;
	ResetSBS1Point : BOOL;
	Reset : BOOL;
	BagSettled : BOOL;
	O_OpenBufferStop : BOOL;
	BagSettledET : UDINT;
	ResetET : UDINT;
END_VAR
```

#### 12_sp2Cyclic.ab
```automation-basic
PROGRAM _CYCLIC
	(* cyclic program *)

;---------------------------------------
;Sequence 12 - SP2 Single point 2 D[912]
;---------------------------------------

;Inputs

I_BagAtBufferStop      = X[8].X03

Enable.BSN[1]			= FALSE	;XA01 Changed from single bag buffer
O_OpenBufferStop   = FALSE

Alarm[15].Name 			= 0
Alarm[15].Bag			= 10003
Alarm[15].Beacon		= TRUE
Alarm[15].Extra			= 0
Alarm[15].Time			= 3000

;Setup Sequence
STEP = D[915]
;Setup Pulse contact
PLS = (STEP <> LASTSTEP)
LASTSTEP = STEP

;Sequence
;Step 0 - Disabled
IF (STEP = 0) THEN
	;Disabled
ENDIF

;Step 1 - check bag stacker calling for bag and empty ready in SIC 3 or SVC5
TON_10ms((STEP=1),300,Reset,ResetET)
IF (STEP = 1) THEN
	D[38] = 0
	ResetSBS1Point = TRUE
	IF Reset THEN
		D[915] = 2
	ENDIF
	ELSE
		ResetSBS1Point = FALSE
ENDIF

;Step 2 - Select SVC5
TON_10ms((I_BagAtBufferStop),200,BagSettled,BagSettledET)
IF (STEP = 2) THEN
	IF BagSettled THEN
		IF Line[25].Clear  AND (D[12]>0)THEN
			D[38] = 1
			C[25] = 0
			D[915] = 3
		ELSE IF (Request.BSN[1] = TRUE) AND (D[18]>0)THEN
			D[38] = 2
			D[915] = 4
		ENDIF
	ENDIF
	;Alarm[27].Name = almBagNotArrived
ENDIF

;select SIC 3
IF (STEP = 3) THEN
O_OpenBufferStop = TRUE
	;IF (D[38] = 1) THEN
		;wait for bag on bypassline
		IF Line[25].Trip THEN
			D[915] = 1
		ENDIF
	;ELSE IF (D[38] = 2) THEN
	;	Enable.BSN[1] = TRUE
		;wait for bag at sbs 1
	;	IF NOT Request.BSN[1] THEN
	;		D[915] = 1
	;	ENDIF
	;ENDIF
	Alarm[15].Name = almBagNotArrived
ENDIF

IF (STEP = 4) THEN
O_OpenBufferStop = TRUE
Enable.BSN[1] = TRUE
	IF NOT Request.BSN[1] THEN
			D[915] = 1
	ENDIF
Alarm[15].Name = almBagNotArrived
ENDIF

;Alarms
TimerAlarm.IN 	= NOT PLS AND (Alarm[15].Name > 0)
TimerAlarm.PT 	= Alarm[15].Time
TimerAlarm FUB TON_10ms()
Alarm[15].On 	= TimerAlarm.Q
Alarm[15].ET 	= TimerAlarm.ET

;Outputs
Y[8].Y03 = O_OpenBufferStop

Y[7].Y14 = ResetSBS1Point

END_PROGRAM
```

### Program Logical/Sequences/10ms/16_sp5 (IEC) - * SP2 Empty bags from SDC1/2

#### 12_sp2.var
```iecst
VAR RETAIN
	STEP : UINT;
	PLS : BOOL;
	LASTSTEP : UINT;
END_VAR
VAR
	TimerAlarm : TON_10ms;
	I_BagAtBuffer : BOOL;
	O_OpenBuffer : BOOL;
	SDC2BufferFullET : TIME;
	SDC2BufferFull : BOOL;
	SettledBufferET : TIME;
	SettledBuffer : BOOL;
	O_OpenSP2BufferStop : BOOL;
	O_SelectPoint : BOOL;
	SP2BufferFull : BOOL;
	SP2BufferFullET : UDINT;
	ParingLoopEnabled : BOOL;
	BagInLoopHasDest : BOOL;
	O_OpenSDC1BufferStop : BOOL;
	BagSettledAtBuffer : BOOL;
	BagSettledAtBufferET : UDINT;
	Alternator : USINT;
	I_OnLineA : BOOL;
	I_TiltA : BOOL;
	I_TiltB : BOOL;
	I_Bagout : BOOL;
	O_OpenBufferStop : BOOL;
	O_SelectLineA : BOOL;
	O_SelectLineB : BOOL;
	O_OpenStops : BOOL;
	O_TiltCylinder : BOOL;
	O_OperatePusher : BOOL;
	PointReset : BOOL;
	PointResetET : UDINT;
	BagAtTilt : BOOL;
	BagAtTiltET : UDINT;
	TiltDown : BOOL;
	TiltDownET : UDINT;
	TiltUp : BOOL;
	TiltUpET : UDINT;
	NotFull : BOOL;
	NotFullET : UDINT;
	Pushed : BOOL;
	SBSN1 : BOOL;
	SBSN1ET : UDINT;
	RequirePusherET : UDINT;
	PushedET : UDINT;
	I_BagAtBufferStop : BOOL;
	O_SP7ToSVC1 : BOOL;
	O_SP7ToSIC3 : BOOL;
	SDC1EmptyBufferFull : BOOL;
	SDC1EmptyBufferFullET : UDINT;
	Reset : BOOL;
	ResetET : UDINT;
	ResetPoint : BOOL;
	I_BagAtSBSF1BufferStop : BOOL;
	I_BagAtExpressBufferStop : BOOL;
	O_OpenBufferStopSBSF1 : BOOL;
	O_OpenBufferStopExpress1 : BOOL;
	BagSettledSBSF1 : BOOL;
	BagSettledSBSF1ET : UDINT;
	BagSettledExpress : BOOL;
	BagSettledExpressET : UDINT;
END_VAR
```

#### 12_sp2Cyclic.ab
```automation-basic
PROGRAM _CYCLIC
	(* cyclic program *)

;---------------------------------------
;Sequence 12 - SP2 Single point 2 D[912]
;---------------------------------------

;Inputs

I_BagAtSBSF1BufferStop   = X[8].X08
I_BagAtExpressBufferStop = X[8].X06

O_OpenBufferStopSBSF1    = FALSE ;Y808
O_OpenBufferStopExpress1 = FALSE ;Y806

Alarm[16].Name 			= 0
Alarm[16].Bag			= 10009
Alarm[16].Beacon		= TRUE
Alarm[16].Extra			= 0
Alarm[16].Time			= 3000

;Setup Sequence
STEP = D[916]
;Setup Pulse contact
PLS = (STEP <> LASTSTEP)
LASTSTEP = STEP

;Sequence
;Step 0 - Disabled
IF (STEP = 0) THEN
	;Disabled
ENDIF

;reset points
TON_10ms((STEP = 1),100,Reset,ResetET)
IF (STEP = 1) THEN
	D[42] = 0

	IF (Reset = TRUE)THEN
		D[916] = 2
	ENDIF
ENDIF

;bag at buffer and send to express or bagstacker
TON_10ms((I_BagAtSBSF1BufferStop),200,BagSettledSBSF1,BagSettledSBSF1ET)
TON_10ms((I_BagAtExpressBufferStop),200,BagSettledExpress,BagSettledExpressET)
IF (STEP = 2) THEN
	IF Line[26].Clear THEN
		IF BagSettledExpress THEN
			D[42]  = 1
			C[26]  = 0
			D[916] = 3
		ELSE IF BagSettledSBSF1 THEN
			D[42]  = 2
			C[26]  = 0
			D[916] = 3
	    ENDIF
	ENDIF
ENDIF

;wait for bag to arrive at destination
IF (STEP = 3) THEN
	IF (D[42] = 1) THEN
		O_OpenBufferStopExpress1 = TRUE
	ELSE IF (D[42] = 2) THEN
		O_OpenBufferStopSBSF1 = TRUE
		;wait for bag at sbs 1
	ENDIF
	IF Line[26].Trip THEN
			D[916] = 1
	ENDIF
ENDIF

;Alarms
TimerAlarm.IN 	= NOT PLS AND (Alarm[16].Name > 0)
TimerAlarm.PT 	= Alarm[16].Time
TimerAlarm FUB TON_10ms()
Alarm[16].On 	= TimerAlarm.Q
Alarm[16].ET 	= TimerAlarm.ET

;Outputs
Y[8].Y06 = (D[42] = 1)
Y[8].Y08 = (D[42] = 2)
END_PROGRAM
```

### Program Logical/Sequences/10ms/17_sic_1 (IEC) - * SP2 Empty bags from SDC1/2

#### 12_sp2.var
```iecst
VAR RETAIN
	STEP : UINT;
	PLS : BOOL;
	LASTSTEP : UINT;
END_VAR
VAR
	TimerAlarm : TON_10ms;
	I_BagAtBuffer : BOOL;
	O_OpenBuffer : BOOL;
	SDC2BufferFullET : TIME;
	SDC2BufferFull : BOOL;
	SettledBufferET : TIME;
	SettledBuffer : BOOL;
	O_OpenSP2BufferStop : BOOL;
	O_SelectPoint : BOOL;
	SP2BufferFull : BOOL;
	SP2BufferFullET : UDINT;
	ParingLoopEnabled : BOOL;
	BagInLoopHasDest : BOOL;
	O_OpenSDC1BufferStop : BOOL;
	BagSettledAtBuffer : BOOL;
	BagSettledAtBufferET : UDINT;
	Alternator : USINT;
	I_PaddleInPosition : BOOL;
	I_BagInIncline : BOOL;
	O_OpenBufferStop : BOOL;
	O_RunMotor : BOOL;
	I_BagAtOutgoingBuffer : BOOL;
	O_OutgoingBufferOpen : BOOL;
	BagSettled : BOOL;
	BagSettledET : UDINT;
	BagNearTop : BOOL;
	BagNearTopET : UDINT;
	CloseBufferStop : BOOL;
	CloseBufferStopET : UDINT;
	RunOn : BOOL;
	RunOnET : UDINT;
	I_BagOutAtTop : BOOL;
	BagAtBuffer : BOOL;
	BagAtBufferET : UDINT;
	I_BagStackerNearFull : BOOL;
	BagStackerHasSpace : BOOL;
	BagStackerHasSpaceET : UDINT;
	SIC3BufferFull : BOOL;
	SIC3BufferFullET : UDINT;
	InclineEnable : BOOL;
END_VAR
```
